Universal Robots PolyScope program: 1_dragon.urp

Program 1_dragon (installation=default directory=/programs/dragon_new createdIn=5.11.9.1010452 lastSavedIn=5.11.9.1010452 robotSerialNumber=20225200364)
Calibrated DH parameters: a=[0.00002, -0.569483, -0.54992, -0.00001, -0.000036, 0]; d=[0.180894, -146.691669, 192.918669, -46.053088, 0.119778, 0.115602]; alpha=[1.571425, -0.001534, 0.003359, 1.568739, -1.571477, 0]; deltaTheta=[0, 0.376258, -0.101074, -0.275185, -0.000002, 0]
Robot Program (runOnlyOnce=false)
  Script file /programs/usbdisk/1/dragon_rotate/john_midlower_rotate.script
    | def azat_dragon_rotate():
    |   # Global parameters:
    |   global speed_ms    = 0.3
    |   global speed_rads  = 0.750
    |   global accel_mss   = 1.000
    |   global accel_radss = 1.200
    |   global blend_radius_m = 0.001
    |   global ref_frame = p[0,0,0,0,0,0]
    | 
    |   #
    |   # TO REMOVE HEADER:
    |   # Go to "Program" -> "Post-Processor Editor"
    |   # Select "Universal Robots"
    |   # Set "INCLUDE_HEADER" to "False"
    |   #
    |   #--------------------------
    |   # Add any default subprograms here
    |   # For example, to drive a gripper as a program call:
    |   # def Gripper_Open():
    |   #   ...
    |   # end
    |   #
    |   # Example to drive a spray gun:
    |   def SprayOn(value):
    |     # use the value as an output:
    |     DO_SPRAY = 5
    |     if value == 0:
    |       set_standard_digital_out(DO_SPRAY, False)
    |     else:
    |       set_standard_digital_out(DO_SPRAY, True)
    |     end
    |   end
    | 
    |   # Example to drive an extruder:
    |   def Extruder(value):
    |     # use the value as an output:
    |     if value < 0:
    |       # stop extruder
    |     else:
    |       # start extruder
    |     end
    |   end
    | 
    |   # Example to move an external axis
    |   def MoveAxis(value):
    |     # use the value as an output:
    |     DO_AXIS_1 = 1
    |     DI_AXIS_1 = 1
    |     if value <= 0:
    |       set_standard_digital_out(DO_AXIS_1, False)
    | 
    |       # Wait for digital input to change state
    |       #while (get_standard_digital_in(DI_AXIS_1) != False):
    |       #  sync()
    |       #end
    |     else:
    |       set_standard_digital_out(DO_AXIS_1, True)
    | 
    |       # Wait for digital input to change state
    |       #while (get_standard_digital_in(DI_AXIS_1) != True):
    |       #  sync()
    |       #end
    |     end
    |   end
    |   #--------------------------
    | 
    | 
    |   # Main program:
    |   # Program generated by RoboDK v5.7.4 for UR10e on 14/08/2024 10:25:34
    |   # Using nominal kinematics.
    |   blend_radius_m = 0.001
    |   speed_ms    = 1.000
    |   ref_frame = p[0.339429, -0.052043, 0.008200, 0.000000, 0.000000, 0.000000]
    |   set_tcp(p[0.000000, 0.000000, 0.252000, 0.000000, 0.000000, 0.000000])
    |   # Show Tool
    |   movej([0.421631, -1.076921, -2.495001, -1.140464, 1.570796, 1.992433],accel_radss,speed_rads,0,0)
    |   movel(pose_trans(ref_frame,p[0.050000, 0.035848, 0.005000, -0.000000, 3.141593, -0.000000]),accel_mss,speed_ms,0,0) # end trace
    |   speed_ms    = 0.002
    |   movel(pose_trans(ref_frame,p[0.050000, 0.035848, -0.000125, -0.000000, 3.141593, -0.000000]),accel_mss,speed_ms,0,0) # end trace
    |   speed_ms    = 0.007
    |   movel(pose_trans(ref_frame,p[0.048115, 0.040844, -0.000125, 0.000000, 3.141593, 0.000000]),accel_mss,speed_ms,0,0.001)
    |   movel(pose_trans(ref_frame,p[0.048793, 0.046214, -0.000125, -0.000000, 3.141593, -0.000000]),accel_mss,speed_ms,0,0.001)
    |   movel(pose_trans(ref_frame,p[0.049357, 0.045822, -0.000125, -0.000000, 3.141593, -0.000000]),accel_mss,speed_ms,0,0.001)
    |   movel(pose_trans(ref_frame,p[0.050418, 0.046022, -0.000125, 0.000000, 3.141593, -0.000000]),accel_mss,speed_ms,0,0.001)
    |   movel(pose_trans(ref_frame,p[0.050476, 0.047250, -0.000125, 0.000000, 3.141593, -0.000000]),accel_mss,speed_ms,0,0.001)
    |   movel(pose_trans(ref_frame,p[0.050281, 0.048486, -0.000125, -0.000000, 3.141593, -0.000000]),accel_mss,speed_ms,0,0.001)
    |   movel(pose_trans(ref_frame,p[0.050801, 0.052016, -0.000125, -0.000000, 3.141593, -0.000000]),accel_mss,speed_ms,0,0.001)
    |   movel(pose_trans(ref_frame,p[0.052856, 0.054981, -0.000125, 0.000000, 3.141593, -0.000000]),accel_mss,speed_ms,0,0.001)
    |   movel(pose_trans(ref_frame,p[0.052477, 0.053383, -0.000125, 0.000000, 3.141593, -0.000000]),accel_mss,speed_ms,0,0.001)
    |   movel(pose_trans(ref_frame,p[0.053030, 0.051842, -0.000125, 0.000000, 3.141593, 0.000000]),accel_mss,speed_ms,0,0.001)
    |   movel(pose_trans(ref_frame,p[0.053222, 0.051718, -0.000125, 0.000000, 3.141593, -0.000000]),accel_mss,speed_ms,0,0.001)
    |   movel(pose_trans(ref_frame,p[0.053441, 0.051660, -0.000125, 0.000000, 3.141593, -0.000000]),accel_mss,speed_ms,0,0.001)
    |   movel(pose_trans(ref_frame,p[0.053830, 0.051770, -0.000125, -0.000000, 3.141593, -0.000000]),accel_mss,speed_ms,0,0.001)
    |   movel(pose_trans(ref_frame,p[0.054167, 0.052030, -0.000125, 0.000000, 3.141593, 0.000000]),accel_mss,speed_ms,0,0.001)
    |   movel(pose_trans(ref_frame,p[0.057601, 0.053765, -0.000125, 0.000000, 3.141593, -0.000000]),accel_mss,speed_ms,0,0.001)
    |   movel(pose_trans(ref_frame,p[0.061373, 0.053375, -0.000125, 0.000000, 3.141593, -0.000000]),accel_mss,speed_ms,0,0.001)
    |   movel(pose_trans(ref_frame,p[0.059629, 0.053360, -0.000125, -0.000000, 3.141593, -0.000000]),accel_mss,speed_ms,0,0.001)
    |   movel(pose_trans(ref_frame,p[0.058435, 0.051934, -0.000125, -0.000000, 3.141593, -0.000000]),accel_mss,speed_ms,0,0.001)
    |   movel(pose_trans(ref_frame,p[0.058753, 0.051481, -0.000125, -0.000000, 3.141593, -0.000000]),accel_mss,speed_ms,0,0.001)
    |   movel(pose_trans(ref_frame,p[0.059332, 0.051255, -0.000125, 0.000000, 3.141593, -0.000000]),accel_mss,speed_ms,0,0.001)
    |   movel(pose_trans(ref_frame,p[0.063602, 0.049837, -0.000125, -0.000000, 3.141593, -0.000000]),accel_mss,speed_ms,0,0.001)
    |   movel(pose_trans(ref_frame,p[0.067592, 0.047737, -0.000125, -0.000000, 3.141593, 0.000000]),accel_mss,speed_ms,0,0.001)
    |   movel(pose_trans(ref_frame,p[0.066591, 0.047674, -0.000125, -0.000000, 3.141593, 0.000000]),accel_mss,speed_ms,0,0.001)
    |   movel(pose_trans(ref_frame,p[0.065618, 0.047434, -0.000125, 0.000000, 3.141593, -0.000000]),accel_mss,speed_ms,0,0.001)
    |   movel(pose_trans(ref_frame,p[0.065188, 0.047247, -0.000125, -0.000000, 3.141593, 0.000000]),accel_mss,speed_ms,0,0.001)
    |   movel(pose_trans(ref_frame,p[0.064838, 0.046949, -0.000125, 0.000000, 3.141593, -0.000000]),accel_mss,speed_ms,0,0.001)
    |   movel(pose_trans(ref_frame,p[0.065795, 0.044806, -0.000125, -0.000000, 3.141593, 0.000000]),accel_mss,speed_ms,0,0.001)
    |   movel(pose_trans(ref_frame,p[0.068800, 0.043786, -0.000125, -0.000000, 3.141593, 0.000000]),accel_mss,speed_ms,0,0.001)
    |   movel(pose_trans(ref_frame,p[0.071196, 0.042031, -0.000125, -0.000000, 3.141593, -0.000000]),accel_mss,speed_ms,0,0.001)
    |   movel(pose_trans(ref_frame,p[0.073265, 0.039897, -0.000125, 0.000000, 3.141593, -0.000000]),accel_mss,speed_ms,0,0.001)
    |   movel(pose_trans(ref_frame,p[0.072103, 0.040443, -0.000125, 0.000000, 3.141593, 0.000000]),accel_mss,speed_ms,0,0.001)
    |   movel(pose_trans(ref_frame,p[0.070839, 0.040620, -0.000125, -0.000000, 3.141593, 0.000000]),accel_mss,speed_ms,0,0.001)
    |   movel(pose_trans(ref_frame,p[0.070205, 0.040771, -0.000125, 0.000000, 3.141593, -0.000000]),accel_mss,speed_ms,0,0.001)
    |   movel(pose_trans(ref_frame,p[0.069592, 0.040656, -0.000125, -0.000000, 3.141593, -0.000000]),accel_mss,speed_ms,0,0.001)
    |   movel(pose_trans(ref_frame,p[0.069908, 0.038813, -0.000125, -0.000000, 3.141593, 0.000000]),accel_mss,speed_ms,0,0.001)
    |   movel(pose_trans(ref_frame,p[0.071559, 0.038089, -0.000125, -0.000000, 3.141593, -0.000000]),accel_mss,speed_ms,0,0.001)
    |   movel(pose_trans(ref_frame,p[0.074165, 0.036670, -0.000125, -0.000000, 3.141593, 0.000000]),accel_mss,speed_ms,0,0.001)
    |   movel(pose_trans(ref_frame,p[0.076688, 0.035073, -0.000125, -0.000000, 3.141593, -0.000000]),accel_mss,speed_ms,0,0.001)
    |   movel(pose_trans(ref_frame,p[0.077386, 0.034559, -0.000125, -0.000000, 3.141593, -0.000000]),accel_mss,speed_ms,0,0.001)
    |   movel(pose_trans(ref_frame,p[0.077983, 0.033940, -0.000125, -0.000000, 3.141593, -0.000000]),accel_mss,speed_ms,0,0.001)
    |   movel(pose_trans(ref_frame,p[0.078075, 0.033778, -0.000125, 0.000000, 3.141593, -0.000000]),accel_mss,speed_ms,0,0.001)
    |   movel(pose_trans(ref_frame,p[0.078069, 0.033607, -0.000125, -0.000000, 3.141593, -0.000000]),accel_mss,speed_ms,0,0.001)
    |   movel(pose_trans(ref_frame,p[0.075726, 0.034474, -0.000125, -0.000000, 3.141593, -0.000000]),accel_mss,speed_ms,0,0.001)
    |   movel(pose_trans(ref_frame,p[0.073247, 0.033725, -0.000125, 0.000000, 3.141593, 0.000000]),accel_mss,speed_ms,0,0.001)
    |   movel(pose_trans(ref_frame,p[0.073124, 0.033569, -0.000125, -0.000000, 3.141593, -0.000000]),accel_mss,speed_ms,0,0.001)
    |   movel(pose_trans(ref_frame,p[0.073061, 0.033386, -0.000125, -0.000000, 3.141593, -0.000000]),accel_mss,speed_ms,0,0.001)
    |   movel(pose_trans(ref_frame,p[0.073215, 0.033032, -0.000125, -0.000000, 3.141593, -0.000000]),accel_mss,speed_ms,0,0.001)
    |   movel(pose_trans(ref_frame,p[0.073585, 0.032804, -0.000125, -0.000000, 3.141593, -0.000000]),accel_mss,speed_ms,0,0.001)
    |   movel(pose_trans(ref_frame,p[0.077970, 0.030799, -0.000125, 0.000000, 3.141593, -0.000000]),accel_mss,speed_ms,0,0.001)
    |   movel(pose_trans(ref_frame,p[0.081965, 0.028072, -0.000125, -0.000000, 3.141593, 0.000000]),accel_mss,speed_ms,0,0.001)
    |   movel(pose_trans(ref_frame,p[0.080851, 0.028334, -0.000125, -0.000000, 3.141593, -0.000000]),accel_mss,speed_ms,0,0.001)
    |   movel(pose_trans(ref_frame,p[0.079709, 0.028175, -0.000125, -0.000000, 3.141593, 0.000000]),accel_mss,speed_ms,0,0.001)
    |   movel(pose_trans(ref_frame,p[0.079538, 0.027599, -0.000125, 0.000000, 3.141593, -0.000000]),accel_mss,speed_ms,0,0.001)
    |   movel(pose_trans(ref_frame,p[0.080054, 0.027314, -0.000125, -0.000000, 3.141593, 0.000000]),accel_mss,speed_ms,0,0.001)
    |   movel(pose_trans(ref_frame,p[0.081649, 0.027083, -0.000125, 0.000000, 3.141593, -0.000000]),accel_mss,speed_ms,0,0.001)
    |   movel(pose_trans(ref_frame,p[0.083244, 0.026828, -0.000125, 0.000000, 3.141593, 0.000000]),accel_mss,speed_ms,0,0.001)
    |   movel(pose_trans(ref_frame,p[0.085130, 0.026266, -0.000125, -0.000000, 3.141593, -0.000000]),accel_mss,speed_ms,0,0.001)
    |   movel(pose_trans(ref_frame,p[0.086815, 0.025298, -0.000125, -0.000000, 3.141593, -0.000000]),accel_mss,speed_ms,0,0.001)
    |   movel(pose_trans(ref_frame,p[0.085082, 0.025169, -0.000125, -0.000000, 3.141593, -0.000000]),accel_mss,speed_ms,0,0.001)
    |   movel(pose_trans(ref_frame,p[0.083511, 0.024408, -0.000125, -0.000000, 3.141593, -0.000000]),accel_mss,speed_ms,0,0.001)
    |   movel(pose_trans(ref_frame,p[0.084423, 0.023039, -0.000125, -0.000000, 3.141593, -0.000000]),accel_mss,speed_ms,0,0.001)
    |   movel(pose_trans(ref_frame,p[0.086438, 0.023247, -0.000125, -0.000000, 3.141593, -0.000000]),accel_mss,speed_ms,0,0.001)
    |   movel(pose_trans(ref_frame,p[0.087631, 0.023229, -0.000125, -0.000000, 3.141593, -0.000000]),accel_mss,speed_ms,0,0.001)
    |   movel(pose_trans(ref_frame,p[0.088824, 0.023201, -0.000125, 0.000000, 3.141593, 0.000000]),accel_mss,speed_ms,0,0.001)
    |   movel(pose_trans(ref_frame,p[0.090324, 0.022840, -0.000125, 0.000000, 3.141593, -0.000000]),accel_mss,speed_ms,0,0.001)
    |   movel(pose_trans(ref_frame,p[0.091725, 0.022190, -0.000125, -0.000000, 3.141593, -0.000000]),accel_mss,speed_ms,0,0.001)
    |   movel(pose_trans(ref_frame,p[0.090634, 0.022048, -0.000125, -0.000000, 3.141593, -0.000000]),accel_mss,speed_ms,0,0.001)
    |   movel(pose_trans(ref_frame,p[0.089714, 0.021514, -0.000125, -0.000000, 3.141593, -0.000000]),accel_mss,speed_ms,0,0.001)
    |   movel(pose_trans(ref_frame,p[0.089568, 0.021326, -0.000125, -0.000000, 3.141593, -0.000000]),accel_mss,speed_ms,0,0.001)
    |   movel(pose_trans(ref_frame,p[0.089490, 0.021107, -0.000125, 0.000000, 3.141593, -0.000000]),accel_mss,speed_ms,0,0.001)
    |   movel(pose_trans(ref_frame,p[0.089956, 0.020148, -0.000125, -0.000000, 3.141593, 0.000000]),accel_mss,speed_ms,0,0.001)
    |   movel(pose_trans(ref_frame,p[0.090905, 0.019837, -0.000125, -0.000000, 3.141593, -0.000000]),accel_mss,speed_ms,0,0.001)
    |   movel(pose_trans(ref_frame,p[0.093609, 0.020103, -0.000125, -0.000000, 3.141593, -0.000000]),accel_mss,speed_ms,0,0.001)
    |   movel(pose_trans(ref_frame,p[0.096074, 0.021219, -0.000125, -0.000000, 3.141593, -0.000000]),accel_mss,speed_ms,0,0.001)
    |   movel(pose_trans(ref_frame,p[0.095278, 0.019985, -0.000125, -0.000000, 3.141593, -0.000000]),accel_mss,speed_ms,0,0.001)
    |   movel(pose_trans(ref_frame,p[0.096057, 0.018680, -0.000125, 0.000000, 3.141593, 0.000000]),accel_mss,speed_ms,0,0.001)
    |   movel(pose_trans(ref_frame,p[0.097535, 0.018934, -0.000125, -0.000000, 3.141593, 0.000000]),accel_mss,speed_ms,0,0.001)
    |   movel(pose_trans(ref_frame,p[0.098790, 0.019781, -0.000125, 0.000000, 3.141593, -0.000000]),accel_mss,speed_ms,0,0.001)
    |   movel(pose_trans(ref_frame,p[0.100083, 0.020616, -0.000125, 0.000000, 3.141593, -0.000000]),accel_mss,speed_ms,0,0.001)
    |   movel(pose_trans(ref_frame,p[0.101189, 0.021687, -0.000125, -0.000000, 3.141593, -0.000000]),accel_mss,speed_ms,0,0.001)
    |   movel(pose_trans(ref_frame,p[0.101202, 0.020923, -0.000125, -0.000000, 3.141593, -0.000000]),accel_mss,speed_ms,0,0.001)
    |   movel(pose_trans(ref_frame,p[0.101280, 0.020162, -0.000125, -0.000000, 3.141593, -0.000000]),accel_mss,speed_ms,0,0.001)
    |   movel(pose_trans(ref_frame,p[0.101434, 0.019617, -0.000125, -0.000000, 3.141593, 0.000000]),accel_mss,speed_ms,0,0.001)
    |   movel(pose_trans(ref_frame,p[0.101820, 0.019279, -0.000125, -0.000000, 3.141593, 0.000000]),accel_mss,speed_ms,0,0.001)
    |   movel(pose_trans(ref_frame,p[0.103405, 0.020161, -0.000125, -0.000000, 3.141593, -0.000000]),accel_mss,speed_ms,0,0.001)
    |   movel(pose_trans(ref_frame,p[0.103922, 0.021711, -0.000125, -0.000000, 3.141593, 0.000000]),accel_mss,speed_ms,0,0.001)
    |   movel(pose_trans(ref_frame,p[0.104603, 0.023835, -0.000125, -0.000000, 3.141593, 0.000000]),accel_mss,speed_ms,0,0.001)
    |   movel(pose_trans(ref_frame,p[0.105672, 0.025813, -0.000125, 0.000000, 3.141593, -0.000000]),accel_mss,speed_ms,0,0.001)
    |   movel(pose_trans(ref_frame,p[0.106210, 0.023998, -0.000125, 0.000000, 3.141593, -0.000000]),accel_mss,speed_ms,0,0.001)
    |   movel(pose_trans(ref_frame,p[0.106813, 0.023627, -0.000125, -0.000000, 3.141593, 0.000000]),accel_mss,speed_ms,0,0.001)
    |   movel(pose_trans(ref_frame,p[0.107376, 0.023906, -0.000125, 0.000000, 3.141593, 0.000000]),accel_mss,speed_ms,0,0.001)
    |   movel(pose_trans(ref_frame,p[0.107881, 0.025705, -0.000125, -0.000000, 3.141593, -0.000000]),accel_mss,speed_ms,0,0.001)
    |   movel(pose_trans(ref_frame,p[0.107658, 0.028092, -0.000125, -0.000000, 3.141593, -0.000000]),accel_mss,speed_ms,0,0.001)
    |   movel(pose_trans(ref_frame,p[0.107800, 0.030579, -0.000125, -0.000000, 3.141593, -0.000000]),accel_mss,speed_ms,0,0.001)
    |   movel(pose_trans(ref_frame,p[0.109047, 0.029228, -0.000125, -0.000000, 3.141593, -0.000000]),accel_mss,speed_ms,0,0.001)
    |   movel(pose_trans(ref_frame,p[0.110204, 0.030182, -0.000125, -0.000000, 3.141593, -0.000000]),accel_mss,speed_ms,0,0.001)
    |   movel(pose_trans(ref_frame,p[0.109002, 0.033200, -0.000125, -0.000000, 3.141593, -0.000000]),accel_mss,speed_ms,0,0.001)
    |   movel(pose_trans(ref_frame,p[0.107979, 0.036132, -0.000125, -0.000000, 3.141593, 0.000000]),accel_mss,speed_ms,0,0.001)
    |   movel(pose_trans(ref_frame,p[0.108895, 0.035281, -0.000125, -0.000000, 3.141593, -0.000000]),accel_mss,speed_ms,0,0.001)
    |   movel(pose_trans(ref_frame,p[0.110237, 0.035493, -0.000125, -0.000000, 3.141593, -0.000000]),accel_mss,speed_ms,0,0.001)
    |   movel(pose_trans(ref_frame,p[0.110068, 0.037051, -0.000125, 0.000000, 3.141593, 0.000000]),accel_mss,speed_ms,0,0.001)
    |   movel(pose_trans(ref_frame,p[0.109162, 0.038243, -0.000125, -0.000000, 3.141593, -0.000000]),accel_mss,speed_ms,0,0.001)
    |   movel(pose_trans(ref_frame,p[0.108731, 0.039432, -0.000125, 0.000000, 3.141593, -0.000000]),accel_mss,speed_ms,0,0.001)
    |   movel(pose_trans(ref_frame,p[0.108673, 0.040695, -0.000125, 0.000000, 3.141593, -0.000000]),accel_mss,speed_ms,0,0) # end trace
    |   speed_ms    = 1.000
    |   movel(pose_trans(ref_frame,p[0.108673, 0.040695, 0.005000, 0.000000, 3.141593, -0.000000]),accel_mss,speed_ms,0,0.001)
    |   movel(pose_trans(ref_frame,p[0.105336, 0.049069, 0.005000, 0.000000, 3.141593, -0.000000]),accel_mss,speed_ms,0,0) # end trace
    |   speed_ms    = 0.002
    |   movel(pose_trans(ref_frame,p[0.105336, 0.049069, -0.000125, 0.000000, 3.141593, 0.000000]),accel_mss,speed_ms,0,0) # end trace
    |   speed_ms    = 0.007
    |   movel(pose_trans(ref_frame,p[0.100848, 0.047278, -0.000125, 0.000000, 3.141593, -0.000000]),accel_mss,speed_ms,0,0.001)
    |   movel(pose_trans(ref_frame,p[0.096181, 0.046825, -0.000125, -0.000000, 3.141593, -0.000000]),accel_mss,speed_ms,0,0.001)
    |   movel(pose_trans(ref_frame,p[0.092012, 0.048769, -0.000125, -0.000000, 3.141593, 0.000000]),accel_mss,speed_ms,0,0.001)
    |   movel(pose_trans(ref_frame,p[0.090230, 0.052991, -0.000125, -0.000000, 3.141593, 0.000000]),accel_mss,speed_ms,0,0.001)
    |   movel(pose_trans(ref_frame,p[0.090956, 0.059068, -0.000125, -0.000000, 3.141593, -0.000000]),accel_mss,speed_ms,0,0.001)
    |   movel(pose_trans(ref_frame,p[0.093240, 0.064896, -0.000125, -0.000000, 3.141593, -0.000000]),accel_mss,speed_ms,0,0.001)
    |   movel(pose_trans(ref_frame,p[0.093396, 0.065125, -0.000125, -0.000000, 3.141593, -0.000000]),accel_mss,speed_ms,0,0.001)
    |   movel(pose_trans(ref_frame,p[0.093608, 0.065293, -0.000125, -0.000000, 3.141593, -0.000000]),accel_mss,speed_ms,0,0.001)
    |   movel(pose_trans(ref_frame,p[0.094176, 0.065243, -0.000125, -0.000000, 3.141593, -0.000000]),accel_mss,speed_ms,0,0.001)
    |   movel(pose_trans(ref_frame,p[0.094662, 0.064808, -0.000125, 0.000000, 3.141593, 0.000000]),accel_mss,speed_ms,0,0.001)
    |   movel(pose_trans(ref_frame,p[0.095614, 0.063660, -0.000125, 0.000000, 3.141593, 0.000000]),accel_mss,speed_ms,0,0.001)
    |   movel(pose_trans(ref_frame,p[0.100924, 0.056746, -0.000125, 0.000000, 3.141593, -0.000000]),accel_mss,speed_ms,0,0.001)
    |   movel(pose_trans(ref_frame,p[0.105953, 0.049801, -0.000125, -0.000000, 3.141593, -0.000000]),accel_mss,speed_ms,0,0.001)
    |   movel(pose_trans(ref_frame,p[0.105818, 0.049295, -0.000125, 0.000000, 3.141593, 0.000000]),accel_mss,speed_ms,0,0.001)
    |   movel(pose_trans(ref_frame,p[0.105578, 0.049182, -0.000125, -0.000000, 3.141593, -0.000000]),accel_mss,speed_ms,0,0.001)
    |   movel(pose_trans(ref_frame,p[0.105336, 0.049069, -0.000125, 0.000000, 3.141593, 0.000000]),accel_mss,speed_ms,0,0) # end trace
    |   speed_ms    = 1.000
    |   movel(pose_trans(ref_frame,p[0.105336, 0.049069, 0.005000, 0.000000, 3.141593, -0.000000]),accel_mss,speed_ms,0,0.001)
    |   movel(pose_trans(ref_frame,p[0.089633, 0.087186, 0.005000, -0.000000, 3.141593, 0.000000]),accel_mss,speed_ms,0,0) # end trace
    |   speed_ms    = 0.002
    |   movel(pose_trans(ref_frame,p[0.089633, 0.087186, -0.000125, -0.000000, 3.141593, -0.000000]),accel_mss,speed_ms,0,0) # end trace
    |   speed_ms    = 0.007
    |   movel(pose_trans(ref_frame,p[0.091088, 0.088696, -0.000125, -0.000000, 3.141593, 0.000000]),accel_mss,speed_ms,0,0.001)
    |   movel(pose_trans(ref_frame,p[0.092593, 0.090142, -0.000125, 0.000000, 3.141593, 0.000000]),accel_mss,speed_ms,0,0.001)
    |   movel(pose_trans(ref_frame,p[0.093893, 0.091163, -0.000125, 0.000000, 3.141593, 0.000000]),accel_mss,speed_ms,0,0.001)
    |   movel(pose_trans(ref_frame,p[0.095145, 0.092291, -0.000125, -0.000000, 3.141593, 0.000000]),accel_mss,speed_ms,0,0.001)
    |   movel(pose_trans(ref_frame,p[0.096993, 0.095273, -0.000125, -0.000000, 3.141593, 0.000000]),accel_mss,speed_ms,0,0.001)
    |   movel(pose_trans(ref_frame,p[0.098237, 0.098544, -0.000125, -0.000000, 3.141593, 0.000000]),accel_mss,speed_ms,0,0.001)
    |   movel(pose_trans(ref_frame,p[0.098481, 0.099687, -0.000125, 0.000000, 3.141593, -0.000000]),accel_mss,speed_ms,0,0.001)
    |   movel(pose_trans(ref_frame,p[0.098141, 0.100704, -0.000125, -0.000000, 3.141593, -0.000000]),accel_mss,speed_ms,0,0.001)
    |   movel(pose_trans(ref_frame,p[0.097842, 0.100958, -0.000125, -0.000000, 3.141593, -0.000000]),accel_mss,speed_ms,0,0.001)
    |   movel(pose_trans(ref_frame,p[0.097539, 0.101210, -0.000125, 0.000000, 3.141593, 0.000000]),accel_mss,speed_ms,0,0.001)
    |   movel(pose_trans(ref_frame,p[0.097169, 0.102392, -0.000125, 0.000000, 3.141593, -0.000000]),accel_mss,speed_ms,0,0.001)
    |   movel(pose_trans(ref_frame,p[0.097527, 0.103718, -0.000125, -0.000000, 3.141593, 0.000000]),accel_mss,speed_ms,0,0.001)
    |   movel(pose_trans(ref_frame,p[0.096297, 0.103890, -0.000125, -0.000000, 3.141593, 0.000000]),accel_mss,speed_ms,0,0.001)
    |   movel(pose_trans(ref_frame,p[0.095148, 0.103405, -0.000125, -0.000000, 3.141593, -0.000000]),accel_mss,speed_ms,0,0.001)
    |   movel(pose_trans(ref_frame,p[0.093699, 0.102652, -0.000125, 0.000000, 3.141593, 0.000000]),accel_mss,speed_ms,0,0.001)
    |   movel(pose_trans(ref_frame,p[0.092339, 0.101738, -0.000125, -0.000000, 3.141593, 0.000000]),accel_mss,speed_ms,0,0.001)
    |   movel(pose_trans(ref_frame,p[0.084495, 0.094077, -0.000125, 0.000000, 3.141593, -0.000000]),accel_mss,speed_ms,0,0.001)
    |   movel(pose_trans(ref_frame,p[0.078491, 0.084897, -0.000125, -0.000000, 3.141593, 0.000000]),accel_mss,speed_ms,0,0.001)
    |   movel(pose_trans(ref_frame,p[0.076525, 0.081104, -0.000125, 0.000000, 3.141593, 0.000000]),accel_mss,speed_ms,0,0.001)
    |   movel(pose_trans(ref_frame,p[0.074922, 0.077142, -0.000125, -0.000000, 3.141593, -0.000000]),accel_mss,speed_ms,0,0.001)
    |   movel(pose_trans(ref_frame,p[0.074131, 0.071003, -0.000125, -0.000000, 3.141593, -0.000000]),accel_mss,speed_ms,0,0.001)
    |   movel(pose_trans(ref_frame,p[0.072889, 0.069893, -0.000125, -0.000000, 3.141593, -0.000000]),accel_mss,speed_ms,0,0.001)
    |   movel(pose_trans(ref_frame,p[0.072797, 0.069931, -0.000125, 0.000000, 3.141593, -0.000000]),accel_mss,speed_ms,0,0.001)
    |   movel(pose_trans(ref_frame,p[0.072716, 0.069992, -0.000125, 0.000000, 3.141593, -0.000000]),accel_mss,speed_ms,0,0.001)
    |   movel(pose_trans(ref_frame,p[0.071475, 0.071671, -0.000125, -0.000000, 3.141593, -0.000000]),accel_mss,speed_ms,0,0.001)
    |   movel(pose_trans(ref_frame,p[0.070262, 0.073293, -0.000125, 0.000000, 3.141593, 0.000000]),accel_mss,speed_ms,0,0.001)
    |   movel(pose_trans(ref_frame,p[0.068510, 0.073911, -0.000125, 0.000000, 3.141593, 0.000000]),accel_mss,speed_ms,0,0.001)
    |   movel(pose_trans(ref_frame,p[0.066701, 0.073510, -0.000125, 0.000000, 3.141593, 0.000000]),accel_mss,speed_ms,0,0.001)
    |   movel(pose_trans(ref_frame,p[0.064031, 0.071756, -0.000125, 0.000000, 3.141593, 0.000000]),accel_mss,speed_ms,0,0.001)
    |   movel(pose_trans(ref_frame,p[0.061632, 0.069604, -0.000125, 0.000000, 3.141593, -0.000000]),accel_mss,speed_ms,0,0.001)
    |   movel(pose_trans(ref_frame,p[0.058330, 0.065115, -0.000125, -0.000000, 3.141593, -0.000000]),accel_mss,speed_ms,0,0.001)
    |   movel(pose_trans(ref_frame,p[0.057824, 0.059503, -0.000125, 0.000000, 3.141593, 0.000000]),accel_mss,speed_ms,0,0.001)
    |   movel(pose_trans(ref_frame,p[0.060086, 0.058641, -0.000125, 0.000000, 3.141593, 0.000000]),accel_mss,speed_ms,0,0.001)
    |   movel(pose_trans(ref_frame,p[0.062094, 0.060133, -0.000125, 0.000000, 3.141593, 0.000000]),accel_mss,speed_ms,0,0.001)
    |   movel(pose_trans(ref_frame,p[0.064267, 0.062034, -0.000125, 0.000000, 3.141593, -0.000000]),accel_mss,speed_ms,0,0.001)
    |   movel(pose_trans(ref_frame,p[0.066707, 0.063601, -0.000125, 0.000000, 3.141593, -0.000000]),accel_mss,speed_ms,0,0.001)
    |   movel(pose_trans(ref_frame,p[0.067317, 0.063786, -0.000125, -0.000000, 3.141593, -0.000000]),accel_mss,speed_ms,0,0.001)
    |   movel(pose_trans(ref_frame,p[0.067927, 0.063723, -0.000125, 0.000000, 3.141593, -0.000000]),accel_mss,speed_ms,0,0.001)
    |   movel(pose_trans(ref_frame,p[0.068318, 0.063438, -0.000125, -0.000000, 3.141593, -0.000000]),accel_mss,speed_ms,0,0.001)
    |   movel(pose_trans(ref_frame,p[0.068611, 0.063039, -0.000125, -0.000000, 3.141593, -0.000000]),accel_mss,speed_ms,0,0.001)
    |   movel(pose_trans(ref_frame,p[0.069511, 0.061129, -0.000125, 0.000000, 3.141593, -0.000000]),accel_mss,speed_ms,0,0.001)
    |   movel(pose_trans(ref_frame,p[0.070136, 0.059096, -0.000125, -0.000000, 3.141593, -0.000000]),accel_mss,speed_ms,0,0.001)
    |   movel(pose_trans(ref_frame,p[0.071200, 0.054465, -0.000125, -0.000000, 3.141593, 0.000000]),accel_mss,speed_ms,0,0.001)
    |   movel(pose_trans(ref_frame,p[0.072592, 0.049848, -0.000125, 0.000000, 3.141593, -0.000000]),accel_mss,speed_ms,0,0.001)
    |   movel(pose_trans(ref_frame,p[0.074780, 0.046144, -0.000125, -0.000000, 3.141593, -0.000000]),accel_mss,speed_ms,0,0.001)
    |   movel(pose_trans(ref_frame,p[0.078924, 0.047029, -0.000125, -0.000000, 3.141593, -0.000000]),accel_mss,speed_ms,0,0.001)
    |   movel(pose_trans(ref_frame,p[0.078996, 0.048255, -0.000125, 0.000000, 3.141593, 0.000000]),accel_mss,speed_ms,0,0.001)
    |   movel(pose_trans(ref_frame,p[0.078814, 0.049489, -0.000125, -0.000000, 3.141593, -0.000000]),accel_mss,speed_ms,0,0.001)
    |   movel(pose_trans(ref_frame,p[0.079748, 0.069610, -0.000125, -0.000000, 3.141593, -0.000000]),accel_mss,speed_ms,0,0.001)
    |   movel(pose_trans(ref_frame,p[0.089629, 0.087186, -0.000125, 0.000000, 3.141593, 0.000000]),accel_mss,speed_ms,0,0) # end trace
    |   speed_ms    = 1.000
    |   movel(pose_trans(ref_frame,p[0.089633, 0.087186, 0.005000, -0.000000, 3.141593, 0.000000]),accel_mss,speed_ms,0,0.001)
    |   movel(pose_trans(ref_frame,p[0.102749, 0.098109, 0.005000, 0.000000, 3.141593, -0.000000]),accel_mss,speed_ms,0,0) # end trace
    |   speed_ms    = 0.002
    |   movel(pose_trans(ref_frame,p[0.102749, 0.098109, -0.000125, 0.000000, 3.141593, -0.000000]),accel_mss,speed_ms,0,0) # end trace
    |   speed_ms    = 0.007
    |   movel(pose_trans(ref_frame,p[0.100717, 0.101702, -0.000125, 0.000000, 3.141593, 0.000000]),accel_mss,speed_ms,0,0.001)
    |   movel(pose_trans(ref_frame,p[0.100054, 0.105778, -0.000125, 0.000000, 3.141593, -0.000000]),accel_mss,speed_ms,0,0.001)
    |   movel(pose_trans(ref_frame,p[0.100478, 0.105179, -0.000125, -0.000000, 3.141593, 0.000000]),accel_mss,speed_ms,0,0.001)
    |   movel(pose_trans(ref_frame,p[0.100830, 0.104483, -0.000125, 0.000000, 3.141593, -0.000000]),accel_mss,speed_ms,0,0.001)
    |   movel(pose_trans(ref_frame,p[0.103117, 0.102032, -0.000125, -0.000000, 3.141593, 0.000000]),accel_mss,speed_ms,0,0.001)
    |   movel(pose_trans(ref_frame,p[0.106032, 0.100361, -0.000125, -0.000000, 3.141593, 0.000000]),accel_mss,speed_ms,0,0.001)
    |   movel(pose_trans(ref_frame,p[0.107531, 0.101698, -0.000125, -0.000000, 3.141593, -0.000000]),accel_mss,speed_ms,0,0.001)
    |   movel(pose_trans(ref_frame,p[0.106753, 0.104177, -0.000125, -0.000000, 3.141593, 0.000000]),accel_mss,speed_ms,0,0.001)
    |   movel(pose_trans(ref_frame,p[0.107988, 0.102605, -0.000125, 0.000000, 3.141593, 0.000000]),accel_mss,speed_ms,0,0.001)
    |   movel(pose_trans(ref_frame,p[0.109319, 0.101130, -0.000125, -0.000000, 3.141593, 0.000000]),accel_mss,speed_ms,0,0.001)
    |   movel(pose_trans(ref_frame,p[0.112898, 0.098528, -0.000125, -0.000000, 3.141593, 0.000000]),accel_mss,speed_ms,0,0.001)
    |   movel(pose_trans(ref_frame,p[0.116000, 0.095504, -0.000125, -0.000000, 3.141593, 0.000000]),accel_mss,speed_ms,0,0.001)
    |   movel(pose_trans(ref_frame,p[0.115507, 0.097438, -0.000125, -0.000000, 3.141593, 0.000000]),accel_mss,speed_ms,0,0.001)
    |   movel(pose_trans(ref_frame,p[0.114821, 0.099297, -0.000125, 0.000000, 3.141593, -0.000000]),accel_mss,speed_ms,0,0.001)
    |   movel(pose_trans(ref_frame,p[0.116243, 0.097691, -0.000125, 0.000000, 3.141593, -0.000000]),accel_mss,speed_ms,0,0.001)
    |   movel(pose_trans(ref_frame,p[0.117809, 0.096208, -0.000125, 0.000000, 3.141593, -0.000000]),accel_mss,speed_ms,0,0.001)
    |   movel(pose_trans(ref_frame,p[0.119446, 0.093932, -0.000125, 0.000000, 3.141593, -0.000000]),accel_mss,speed_ms,0,0.001)
    |   movel(pose_trans(ref_frame,p[0.120874, 0.091548, -0.000125, 0.000000, 3.141593, 0.000000]),accel_mss,speed_ms,0,0.001)
    |   movel(pose_trans(ref_frame,p[0.121474, 0.090885, -0.000125, 0.000000, 3.141593, -0.000000]),accel_mss,speed_ms,0,0.001)
    |   movel(pose_trans(ref_frame,p[0.122260, 0.090597, -0.000125, -0.000000, 3.141593, 0.000000]),accel_mss,speed_ms,0,0.001)
    |   movel(pose_trans(ref_frame,p[0.123089, 0.090981, -0.000125, 0.000000, 3.141593, -0.000000]),accel_mss,speed_ms,0,0.001)
    |   movel(pose_trans(ref_frame,p[0.123661, 0.091788, -0.000125, 0.000000, 3.141593, -0.000000]),accel_mss,speed_ms,0,0.001)
    |   movel(pose_trans(ref_frame,p[0.124539, 0.088269, -0.000125, -0.000000, 3.141593, 0.000000]),accel_mss,speed_ms,0,0.001)
    |   movel(pose_trans(ref_frame,p[0.125564, 0.084887, -0.000125, -0.000000, 3.141593, -0.000000]),accel_mss,speed_ms,0,0.001)
    |   movel(pose_trans(ref_frame,p[0.125556, 0.082021, -0.000125, -0.000000, 3.141593, 0.000000]),accel_mss,speed_ms,0,0.001)
    |   movel(pose_trans(ref_frame,p[0.124836, 0.079246, -0.000125, -0.000000, 3.141593, -0.000000]),accel_mss,speed_ms,0,0) # end trace
    |   speed_ms    = 1.000
    |   movel(pose_trans(ref_frame,p[0.124836, 0.079246, 0.005000, -0.000000, 3.141593, 0.000000]),accel_mss,speed_ms,0,0.001)
    |   movel(pose_trans(ref_frame,p[0.070961, 0.083800, 0.005000, -0.000000, 3.141593, -0.000000]),accel_mss,speed_ms,0,0) # end trace
    |   speed_ms    = 0.002
    |   movel(pose_trans(ref_frame,p[0.070961, 0.083800, -0.000125, -0.000000, 3.141593, -0.000000]),accel_mss,speed_ms,0,0) # end trace
    |   speed_ms    = 0.007
    |   movel(pose_trans(ref_frame,p[0.069945, 0.082016, -0.000125, -0.000000, 3.141593, -0.000000]),accel_mss,speed_ms,0,0.001)
    |   movel(pose_trans(ref_frame,p[0.068221, 0.080903, -0.000125, -0.000000, 3.141593, -0.000000]),accel_mss,speed_ms,0,0.001)
    |   movel(pose_trans(ref_frame,p[0.062416, 0.082363, -0.000125, 0.000000, 3.141593, -0.000000]),accel_mss,speed_ms,0,0.001)
    |   movel(pose_trans(ref_frame,p[0.059213, 0.087150, -0.000125, 0.000000, 3.141593, 0.000000]),accel_mss,speed_ms,0,0.001)
    |   movel(pose_trans(ref_frame,p[0.057492, 0.092576, -0.000125, 0.000000, 3.141593, 0.000000]),accel_mss,speed_ms,0,0.001)
    |   movel(pose_trans(ref_frame,p[0.056740, 0.098209, -0.000125, -0.000000, 3.141593, 0.000000]),accel_mss,speed_ms,0,0.001)
    |   movel(pose_trans(ref_frame,p[0.056549, 0.100188, -0.000125, -0.000000, 3.141593, -0.000000]),accel_mss,speed_ms,0,0.001)
    |   movel(pose_trans(ref_frame,p[0.056117, 0.102115, -0.000125, 0.000000, 3.141593, 0.000000]),accel_mss,speed_ms,0,0.001)
    |   movel(pose_trans(ref_frame,p[0.055117, 0.104549, -0.000125, -0.000000, 3.141593, 0.000000]),accel_mss,speed_ms,0,0.001)
    |   movel(pose_trans(ref_frame,p[0.054994, 0.106976, -0.000125, -0.000000, 3.141593, -0.000000]),accel_mss,speed_ms,0,0.001)
    |   movel(pose_trans(ref_frame,p[0.054089, 0.104072, -0.000125, -0.000000, 3.141593, -0.000000]),accel_mss,speed_ms,0,0.001)
    |   movel(pose_trans(ref_frame,p[0.053416, 0.101119, -0.000125, 0.000000, 3.141593, -0.000000]),accel_mss,speed_ms,0,0.001)
    |   movel(pose_trans(ref_frame,p[0.052834, 0.097793, -0.000125, -0.000000, 3.141593, -0.000000]),accel_mss,speed_ms,0,0.001)
    |   movel(pose_trans(ref_frame,p[0.052414, 0.094442, -0.000125, 0.000000, 3.141593, -0.000000]),accel_mss,speed_ms,0,0.001)
    |   movel(pose_trans(ref_frame,p[0.052122, 0.091150, -0.000125, -0.000000, 3.141593, -0.000000]),accel_mss,speed_ms,0,0.001)
    |   movel(pose_trans(ref_frame,p[0.052084, 0.087843, -0.000125, 0.000000, 3.141593, 0.000000]),accel_mss,speed_ms,0,0.001)
    |   movel(pose_trans(ref_frame,p[0.052355, 0.085273, -0.000125, -0.000000, 3.141593, -0.000000]),accel_mss,speed_ms,0,0.001)
    |   movel(pose_trans(ref_frame,p[0.052616, 0.082645, -0.000125, 0.000000, 3.141593, 0.000000]),accel_mss,speed_ms,0,0.001)
    |   movel(pose_trans(ref_frame,p[0.052535, 0.081947, -0.000125, -0.000000, 3.141593, 0.000000]),accel_mss,speed_ms,0,0.001)
    |   movel(pose_trans(ref_frame,p[0.052090, 0.081554, -0.000125, 0.000000, 3.141593, -0.000000]),accel_mss,speed_ms,0,0.001)
    |   movel(pose_trans(ref_frame,p[0.051868, 0.081568, -0.000125, -0.000000, 3.141593, -0.000000]),accel_mss,speed_ms,0,0.001)
    |   movel(pose_trans(ref_frame,p[0.051653, 0.081638, -0.000125, -0.000000, 3.141593, -0.000000]),accel_mss,speed_ms,0,0.001)
    |   movel(pose_trans(ref_frame,p[0.044813, 0.088250, -0.000125, 0.000000, 3.141593, 0.000000]),accel_mss,speed_ms,0,0.001)
    |   movel(pose_trans(ref_frame,p[0.041449, 0.096978, -0.000125, -0.000000, 3.141593, 0.000000]),accel_mss,speed_ms,0,0.001)
    |   movel(pose_trans(ref_frame,p[0.041171, 0.097676, -0.000125, 0.000000, 3.141593, -0.000000]),accel_mss,speed_ms,0,0.001)
    |   movel(pose_trans(ref_frame,p[0.040734, 0.098269, -0.000125, 0.000000, 3.141593, 0.000000]),accel_mss,speed_ms,0,0.001)
    |   movel(pose_trans(ref_frame,p[0.038679, 0.098423, -0.000125, 0.000000, 3.141593, 0.000000]),accel_mss,speed_ms,0,0.001)
    |   movel(pose_trans(ref_frame,p[0.037369, 0.097061, -0.000125, -0.000000, 3.141593, 0.000000]),accel_mss,speed_ms,0,0.001)
    |   movel(pose_trans(ref_frame,p[0.036035, 0.094122, -0.000125, 0.000000, 3.141593, -0.000000]),accel_mss,speed_ms,0,0.001)
    |   movel(pose_trans(ref_frame,p[0.035297, 0.090976, -0.000125, 0.000000, 3.141593, 0.000000]),accel_mss,speed_ms,0,0.001)
    |   movel(pose_trans(ref_frame,p[0.035073, 0.089838, -0.000125, -0.000000, 3.141593, 0.000000]),accel_mss,speed_ms,0,0.001)
    |   movel(pose_trans(ref_frame,p[0.034332, 0.088884, -0.000125, 0.000000, 3.141593, 0.000000]),accel_mss,speed_ms,0,0.001)
    |   movel(pose_trans(ref_frame,p[0.033478, 0.088790, -0.000125, -0.000000, 3.141593, 0.000000]),accel_mss,speed_ms,0,0.001)
    |   movel(pose_trans(ref_frame,p[0.032671, 0.089210, -0.000125, 0.000000, 3.141593, 0.000000]),accel_mss,speed_ms,0,0.001)
    |   movel(pose_trans(ref_frame,p[0.031591, 0.090296, -0.000125, -0.000000, 3.141593, -0.000000]),accel_mss,speed_ms,0,0.001)
    |   movel(pose_trans(ref_frame,p[0.030677, 0.091522, -0.000125, 0.000000, 3.141593, 0.000000]),accel_mss,speed_ms,0,0.001)
    |   movel(pose_trans(ref_frame,p[0.029076, 0.096690, -0.000125, 0.000000, 3.141593, -0.000000]),accel_mss,speed_ms,0,0.001)
    |   movel(pose_trans(ref_frame,p[0.029868, 0.101986, -0.000125, 0.000000, 3.141593, 0.000000]),accel_mss,speed_ms,0,0.001)
    |   movel(pose_trans(ref_frame,p[0.031346, 0.105758, -0.000125, 0.000000, 3.141593, 0.000000]),accel_mss,speed_ms,0,0.001)
    |   movel(pose_trans(ref_frame,p[0.033747, 0.109039, -0.000125, -0.000000, 3.141593, -0.000000]),accel_mss,speed_ms,0,0.001)
    |   movel(pose_trans(ref_frame,p[0.036020, 0.110818, -0.000125, -0.000000, 3.141593, -0.000000]),accel_mss,speed_ms,0,0.001)
    |   movel(pose_trans(ref_frame,p[0.038929, 0.111276, -0.000125, -0.000000, 3.141593, -0.000000]),accel_mss,speed_ms,0,0.001)
    |   movel(pose_trans(ref_frame,p[0.041535, 0.109044, -0.000125, -0.000000, 3.141593, 0.000000]),accel_mss,speed_ms,0,0.001)
    |   movel(pose_trans(ref_frame,p[0.042762, 0.105959, -0.000125, 0.000000, 3.141593, 0.000000]),accel_mss,speed_ms,0,0.001)
    |   movel(pose_trans(ref_frame,p[0.043328, 0.104611, -0.000125, 0.000000, 3.141593, -0.000000]),accel_mss,speed_ms,0,0.001)
    |   movel(pose_trans(ref_frame,p[0.044464, 0.103624, -0.000125, 0.000000, 3.141593, 0.000000]),accel_mss,speed_ms,0,0.001)
    |   movel(pose_trans(ref_frame,p[0.044178, 0.104207, -0.000125, -0.000000, 3.141593, 0.000000]),accel_mss,speed_ms,0,0.001)
    |   movel(pose_trans(ref_frame,p[0.045734, 0.107913, -0.000125, -0.000000, 3.141593, -0.000000]),accel_mss,speed_ms,0,0.001)
    |   movel(pose_trans(ref_frame,p[0.047715, 0.111798, -0.000125, -0.000000, 3.141593, -0.000000]),accel_mss,speed_ms,0,0.001)
    |   movel(pose_trans(ref_frame,p[0.048146, 0.112505, -0.000125, 0.000000, 3.141593, -0.000000]),accel_mss,speed_ms,0,0.001)
    |   movel(pose_trans(ref_frame,p[0.050447, 0.115705, -0.000125, -0.000000, 3.141593, -0.000000]),accel_mss,speed_ms,0,0.001)
    |   movel(pose_trans(ref_frame,p[0.052920, 0.118790, -0.000125, -0.000000, 3.141593, -0.000000]),accel_mss,speed_ms,0,0.001)
    |   movel(pose_trans(ref_frame,p[0.055404, 0.121521, -0.000125, -0.000000, 3.141593, 0.000000]),accel_mss,speed_ms,0,0.001)
    |   movel(pose_trans(ref_frame,p[0.058393, 0.123580, -0.000125, -0.000000, 3.141593, 0.000000]),accel_mss,speed_ms,0,0.001)
    |   movel(pose_trans(ref_frame,p[0.058302, 0.121953, -0.000125, -0.000000, 3.141593, -0.000000]),accel_mss,speed_ms,0,0.001)
    |   movel(pose_trans(ref_frame,p[0.058332, 0.121467, -0.000125, -0.000000, 3.141593, -0.000000]),accel_mss,speed_ms,0,0.001)
    |   movel(pose_trans(ref_frame,p[0.058594, 0.121121, -0.000125, 0.000000, 3.141593, -0.000000]),accel_mss,speed_ms,0,0.001)
    |   movel(pose_trans(ref_frame,p[0.058956, 0.121095, -0.000125, -0.000000, 3.141593, -0.000000]),accel_mss,speed_ms,0,0.001)
    |   movel(pose_trans(ref_frame,p[0.059323, 0.121228, -0.000125, 0.000000, 3.141593, 0.000000]),accel_mss,speed_ms,0,0.001)
    |   movel(pose_trans(ref_frame,p[0.060345, 0.121460, -0.000125, -0.000000, 3.141593, -0.000000]),accel_mss,speed_ms,0,0.001)
    |   movel(pose_trans(ref_frame,p[0.061388, 0.121359, -0.000125, 0.000000, 3.141593, -0.000000]),accel_mss,speed_ms,0,0.001)
    |   movel(pose_trans(ref_frame,p[0.061473, 0.121332, -0.000125, 0.000000, 3.141593, 0.000000]),accel_mss,speed_ms,0,0.001)
    |   movel(pose_trans(ref_frame,p[0.061545, 0.121284, -0.000125, 0.000000, 3.141593, -0.000000]),accel_mss,speed_ms,0,0.001)
    |   movel(pose_trans(ref_frame,p[0.061575, 0.121024, -0.000125, 0.000000, 3.141593, -0.000000]),accel_mss,speed_ms,0,0.001)
    |   movel(pose_trans(ref_frame,p[0.061474, 0.120721, -0.000125, 0.000000, 3.141593, -0.000000]),accel_mss,speed_ms,0,0.001)
    |   movel(pose_trans(ref_frame,p[0.061582, 0.120424, -0.000125, 0.000000, 3.141593, 0.000000]),accel_mss,speed_ms,0,0.001)
    |   movel(pose_trans(ref_frame,p[0.061883, 0.120274, -0.000125, 0.000000, 3.141593, 0.000000]),accel_mss,speed_ms,0,0.001)
    |   movel(pose_trans(ref_frame,p[0.062212, 0.120291, -0.000125, -0.000000, 3.141593, -0.000000]),accel_mss,speed_ms,0,0.001)
    |   movel(pose_trans(ref_frame,p[0.062533, 0.120391, -0.000125, -0.000000, 3.141593, 0.000000]),accel_mss,speed_ms,0,0.001)
    |   movel(pose_trans(ref_frame,p[0.064505, 0.121106, -0.000125, -0.000000, 3.141593, 0.000000]),accel_mss,speed_ms,0,0.001)
    |   movel(pose_trans(ref_frame,p[0.061922, 0.119266, -0.000125, 0.000000, 3.141593, -0.000000]),accel_mss,speed_ms,0,0.001)
    |   movel(pose_trans(ref_frame,p[0.059801, 0.116874, -0.000125, -0.000000, 3.141593, -0.000000]),accel_mss,speed_ms,0,0.001)
    |   movel(pose_trans(ref_frame,p[0.057879, 0.114087, -0.000125, -0.000000, 3.141593, 0.000000]),accel_mss,speed_ms,0,0.001)
    |   movel(pose_trans(ref_frame,p[0.056438, 0.111016, -0.000125, -0.000000, 3.141593, -0.000000]),accel_mss,speed_ms,0,0.001)
    |   movel(pose_trans(ref_frame,p[0.056309, 0.106637, -0.000125, 0.000000, 3.141593, 0.000000]),accel_mss,speed_ms,0,0.001)
    |   movel(pose_trans(ref_frame,p[0.058011, 0.102615, -0.000125, 0.000000, 3.141593, -0.000000]),accel_mss,speed_ms,0,0.001)
    |   movel(pose_trans(ref_frame,p[0.059784, 0.101649, -0.000125, -0.000000, 3.141593, -0.000000]),accel_mss,speed_ms,0,0.001)
    |   movel(pose_trans(ref_frame,p[0.061498, 0.102733, -0.000125, 0.000000, 3.141593, -0.000000]),accel_mss,speed_ms,0,0.001)
    |   movel(pose_trans(ref_frame,p[0.063515, 0.105687, -0.000125, -0.000000, 3.141593, 0.000000]),accel_mss,speed_ms,0,0.001)
    |   movel(pose_trans(ref_frame,p[0.066545, 0.107663, -0.000125, -0.000000, 3.141593, -0.000000]),accel_mss,speed_ms,0,0.001)
    |   movel(pose_trans(ref_frame,p[0.067506, 0.107818, -0.000125, -0.000000, 3.141593, -0.000000]),accel_mss,speed_ms,0,0.001)
    |   movel(pose_trans(ref_frame,p[0.068490, 0.107788, -0.000125, 0.000000, 3.141593, -0.000000]),accel_mss,speed_ms,0,0.001)
    |   movel(pose_trans(ref_frame,p[0.073823, 0.104642, -0.000125, -0.000000, 3.141593, 0.000000]),accel_mss,speed_ms,0,0.001)
    |   movel(pose_trans(ref_frame,p[0.076606, 0.099224, -0.000125, -0.000000, 3.141593, 0.000000]),accel_mss,speed_ms,0,0.001)
    |   movel(pose_trans(ref_frame,p[0.078349, 0.090265, -0.000125, 0.000000, 3.141593, 0.000000]),accel_mss,speed_ms,0,0.001)
    |   movel(pose_trans(ref_frame,p[0.074472, 0.081840, -0.000125, 0.000000, 3.141593, 0.000000]),accel_mss,speed_ms,0,0.001)
    |   movel(pose_trans(ref_frame,p[0.074097, 0.081567, -0.000125, -0.000000, 3.141593, 0.000000]),accel_mss,speed_ms,0,0.001)
    |   movel(pose_trans(ref_frame,p[0.073668, 0.081424, -0.000125, 0.000000, 3.141593, 0.000000]),accel_mss,speed_ms,0,0.001)
    |   movel(pose_trans(ref_frame,p[0.073028, 0.081623, -0.000125, 0.000000, 3.141593, 0.000000]),accel_mss,speed_ms,0,0.001)
    |   movel(pose_trans(ref_frame,p[0.072580, 0.082171, -0.000125, -0.000000, 3.141593, -0.000000]),accel_mss,speed_ms,0,0.001)
    |   movel(pose_trans(ref_frame,p[0.072124, 0.083674, -0.000125, 0.000000, 3.141593, -0.000000]),accel_mss,speed_ms,0,0.001)
    |   movel(pose_trans(ref_frame,p[0.071925, 0.085234, -0.000125, -0.000000, 3.141593, 0.000000]),accel_mss,speed_ms,0,0.001)
    |   movel(pose_trans(ref_frame,p[0.071809, 0.085506, -0.000125, 0.000000, 3.141593, 0.000000]),accel_mss,speed_ms,0,0.001)
    |   movel(pose_trans(ref_frame,p[0.071555, 0.085629, -0.000125, 0.000000, 3.141593, 0.000000]),accel_mss,speed_ms,0,0.001)
    |   movel(pose_trans(ref_frame,p[0.071311, 0.085120, -0.000125, -0.000000, 3.141593, -0.000000]),accel_mss,speed_ms,0,0.001)
    |   movel(pose_trans(ref_frame,p[0.071102, 0.084572, -0.000125, -0.000000, 3.141593, -0.000000]),accel_mss,speed_ms,0,0.001)
    |   movel(pose_trans(ref_frame,p[0.070576, 0.089151, -0.000125, 0.000000, 3.141593, -0.000000]),accel_mss,speed_ms,0,0.001)
    |   movel(pose_trans(ref_frame,p[0.069756, 0.093688, -0.000125, -0.000000, 3.141593, 0.000000]),accel_mss,speed_ms,0,0.001)
    |   movel(pose_trans(ref_frame,p[0.069243, 0.095663, -0.000125, 0.000000, 3.141593, -0.000000]),accel_mss,speed_ms,0,0.001)
    |   movel(pose_trans(ref_frame,p[0.068151, 0.097410, -0.000125, -0.000000, 3.141593, -0.000000]),accel_mss,speed_ms,0,0.001)
    |   movel(pose_trans(ref_frame,p[0.065563, 0.098071, -0.000125, 0.000000, 3.141593, -0.000000]),accel_mss,speed_ms,0,0.001)
    |   movel(pose_trans(ref_frame,p[0.063250, 0.096920, -0.000125, -0.000000, 3.141593, -0.000000]),accel_mss,speed_ms,0,0) # end trace
    |   speed_ms    = 1.000
    |   movel(pose_trans(ref_frame,p[0.063250, 0.096920, 0.005000, -0.000000, 3.141593, -0.000000]),accel_mss,speed_ms,0,0.001)
    |   movel(pose_trans(ref_frame,p[0.059449, 0.103780, 0.005000, 0.000000, 3.141593, -0.000000]),accel_mss,speed_ms,0,0) # end trace
    |   speed_ms    = 0.002
    |   movel(pose_trans(ref_frame,p[0.059449, 0.103780, -0.000125, 0.000000, 3.141593, -0.000000]),accel_mss,speed_ms,0,0) # end trace
    |   speed_ms    = 0.007
    |   movel(pose_trans(ref_frame,p[0.059380, 0.106675, -0.000125, -0.000000, 3.141593, 0.000000]),accel_mss,speed_ms,0,0.001)
    |   movel(pose_trans(ref_frame,p[0.060031, 0.109497, -0.000125, 0.000000, 3.141593, 0.000000]),accel_mss,speed_ms,0,0.001)
    |   movel(pose_trans(ref_frame,p[0.059947, 0.108523, -0.000125, 0.000000, 3.141593, -0.000000]),accel_mss,speed_ms,0,0.001)
    |   movel(pose_trans(ref_frame,p[0.060044, 0.107597, -0.000125, 0.000000, 3.141593, 0.000000]),accel_mss,speed_ms,0,0.001)
    |   movel(pose_trans(ref_frame,p[0.060430, 0.107054, -0.000125, -0.000000, 3.141593, -0.000000]),accel_mss,speed_ms,0,0.001)
    |   movel(pose_trans(ref_frame,p[0.061164, 0.107254, -0.000125, 0.000000, 3.141593, -0.000000]),accel_mss,speed_ms,0,0.001)
    |   movel(pose_trans(ref_frame,p[0.061898, 0.109971, -0.000125, -0.000000, 3.141593, 0.000000]),accel_mss,speed_ms,0,0.001)
    |   movel(pose_trans(ref_frame,p[0.063165, 0.112630, -0.000125, -0.000000, 3.141593, -0.000000]),accel_mss,speed_ms,0,0.001)
    |   movel(pose_trans(ref_frame,p[0.062963, 0.111210, -0.000125, 0.000000, 3.141593, -0.000000]),accel_mss,speed_ms,0,0.001)
    |   movel(pose_trans(ref_frame,p[0.064114, 0.110458, -0.000125, 0.000000, 3.141593, -0.000000]),accel_mss,speed_ms,0,0.001)
    |   movel(pose_trans(ref_frame,p[0.065053, 0.111647, -0.000125, -0.000000, 3.141593, 0.000000]),accel_mss,speed_ms,0,0.001)
    |   movel(pose_trans(ref_frame,p[0.066021, 0.112722, -0.000125, 0.000000, 3.141593, -0.000000]),accel_mss,speed_ms,0,0) # end trace
    |   speed_ms    = 1.000
    |   movel(pose_trans(ref_frame,p[0.066021, 0.112722, 0.005000, 0.000000, 3.141593, 0.000000]),accel_mss,speed_ms,0,0.001)
    |   movel(pose_trans(ref_frame,p[0.063840, 0.108129, 0.005000, -0.000000, 3.141593, 0.000000]),accel_mss,speed_ms,0,0) # end trace
    |   speed_ms    = 0.002
    |   movel(pose_trans(ref_frame,p[0.063840, 0.108129, -0.000125, -0.000000, 3.141593, 0.000000]),accel_mss,speed_ms,0,0) # end trace
    |   speed_ms    = 0.007
    |   movel(pose_trans(ref_frame,p[0.064907, 0.109512, -0.000125, 0.000000, 3.141593, 0.000000]),accel_mss,speed_ms,0,0.001)
    |   movel(pose_trans(ref_frame,p[0.065896, 0.110959, -0.000125, -0.000000, 3.141593, 0.000000]),accel_mss,speed_ms,0,0.001)
    |   movel(pose_trans(ref_frame,p[0.067070, 0.112271, -0.000125, 0.000000, 3.141593, 0.000000]),accel_mss,speed_ms,0,0.001)
    |   movel(pose_trans(ref_frame,p[0.068564, 0.113135, -0.000125, -0.000000, 3.141593, 0.000000]),accel_mss,speed_ms,0,0.001)
    |   movel(pose_trans(ref_frame,p[0.067195, 0.112039, -0.000125, -0.000000, 3.141593, -0.000000]),accel_mss,speed_ms,0,0.001)
    |   movel(pose_trans(ref_frame,p[0.068061, 0.110419, -0.000125, -0.000000, 3.141593, 0.000000]),accel_mss,speed_ms,0,0.001)
    |   movel(pose_trans(ref_frame,p[0.068442, 0.110479, -0.000125, 0.000000, 3.141593, 0.000000]),accel_mss,speed_ms,0,0.001)
    |   movel(pose_trans(ref_frame,p[0.068805, 0.110635, -0.000125, 0.000000, 3.141593, -0.000000]),accel_mss,speed_ms,0,0.001)
    |   movel(pose_trans(ref_frame,p[0.071290, 0.111502, -0.000125, -0.000000, 3.141593, 0.000000]),accel_mss,speed_ms,0,0.001)
    |   movel(pose_trans(ref_frame,p[0.073921, 0.110990, -0.000125, 0.000000, 3.141593, 0.000000]),accel_mss,speed_ms,0,0.001)
    |   movel(pose_trans(ref_frame,p[0.072888, 0.111019, -0.000125, -0.000000, 3.141593, 0.000000]),accel_mss,speed_ms,0,0.001)
    |   movel(pose_trans(ref_frame,p[0.072031, 0.110400, -0.000125, -0.000000, 3.141593, -0.000000]),accel_mss,speed_ms,0,0.001)
    |   movel(pose_trans(ref_frame,p[0.072094, 0.109682, -0.000125, -0.000000, 3.141593, 0.000000]),accel_mss,speed_ms,0,0.001)
    |   movel(pose_trans(ref_frame,p[0.072833, 0.109390, -0.000125, 0.000000, 3.141593, 0.000000]),accel_mss,speed_ms,0,0.001)
    |   movel(pose_trans(ref_frame,p[0.075064, 0.108702, -0.000125, -0.000000, 3.141593, -0.000000]),accel_mss,speed_ms,0,0.001)
    |   movel(pose_trans(ref_frame,p[0.076943, 0.107272, -0.000125, -0.000000, 3.141593, -0.000000]),accel_mss,speed_ms,0,0.001)
    |   movel(pose_trans(ref_frame,p[0.076310, 0.107481, -0.000125, 0.000000, 3.141593, -0.000000]),accel_mss,speed_ms,0,0.001)
    |   movel(pose_trans(ref_frame,p[0.075606, 0.107337, -0.000125, 0.000000, 3.141593, -0.000000]),accel_mss,speed_ms,0,0.001)
    |   movel(pose_trans(ref_frame,p[0.075974, 0.105904, -0.000125, -0.000000, 3.141593, -0.000000]),accel_mss,speed_ms,0,0.001)
    |   movel(pose_trans(ref_frame,p[0.078068, 0.104825, -0.000125, 0.000000, 3.141593, 0.000000]),accel_mss,speed_ms,0,0.001)
    |   movel(pose_trans(ref_frame,p[0.079129, 0.103687, -0.000125, -0.000000, 3.141593, 0.000000]),accel_mss,speed_ms,0,0.001)
    |   movel(pose_trans(ref_frame,p[0.079839, 0.102325, -0.000125, 0.000000, 3.141593, -0.000000]),accel_mss,speed_ms,0,0.001)
    |   movel(pose_trans(ref_frame,p[0.079361, 0.102884, -0.000125, 0.000000, 3.141593, -0.000000]),accel_mss,speed_ms,0,0.001)
    |   movel(pose_trans(ref_frame,p[0.078697, 0.103214, -0.000125, -0.000000, 3.141593, 0.000000]),accel_mss,speed_ms,0,0.001)
    |   movel(pose_trans(ref_frame,p[0.078265, 0.102978, -0.000125, -0.000000, 3.141593, -0.000000]),accel_mss,speed_ms,0,0.001)
    |   movel(pose_trans(ref_frame,p[0.078248, 0.102478, -0.000125, 0.000000, 3.141593, -0.000000]),accel_mss,speed_ms,0,0.001)
    |   movel(pose_trans(ref_frame,p[0.079358, 0.099460, -0.000125, 0.000000, 3.141593, -0.000000]),accel_mss,speed_ms,0,0.001)
    |   movel(pose_trans(ref_frame,p[0.079740, 0.096188, -0.000125, -0.000000, 3.141593, -0.000000]),accel_mss,speed_ms,0,0) # end trace
    |   speed_ms    = 1.000
    |   movel(pose_trans(ref_frame,p[0.079740, 0.096188, 0.005000, -0.000000, 3.141593, 0.000000]),accel_mss,speed_ms,0,0.001)
    |   movel(pose_trans(ref_frame,p[0.069434, 0.088428, 0.005000, -0.000000, 3.141593, -0.000000]),accel_mss,speed_ms,0,0) # end trace
    |   speed_ms    = 0.002
    |   movel(pose_trans(ref_frame,p[0.069434, 0.088428, -0.000125, -0.000000, 3.141593, 0.000000]),accel_mss,speed_ms,0,0) # end trace
    |   speed_ms    = 0.007
    |   movel(pose_trans(ref_frame,p[0.068644, 0.086784, -0.000125, 0.000000, 3.141593, 0.000000]),accel_mss,speed_ms,0,0.001)
    |   movel(pose_trans(ref_frame,p[0.066902, 0.086088, -0.000125, 0.000000, 3.141593, -0.000000]),accel_mss,speed_ms,0,0.001)
    |   movel(pose_trans(ref_frame,p[0.064540, 0.087037, -0.000125, 0.000000, 3.141593, -0.000000]),accel_mss,speed_ms,0,0.001)
    |   movel(pose_trans(ref_frame,p[0.063232, 0.089163, -0.000125, -0.000000, 3.141593, 0.000000]),accel_mss,speed_ms,0,0.001)
    |   movel(pose_trans(ref_frame,p[0.063410, 0.093674, -0.000125, -0.000000, 3.141593, -0.000000]),accel_mss,speed_ms,0,0.001)
    |   movel(pose_trans(ref_frame,p[0.066314, 0.097161, -0.000125, -0.000000, 3.141593, 0.000000]),accel_mss,speed_ms,0,0) # end trace
    |   speed_ms    = 1.000
    |   movel(pose_trans(ref_frame,p[0.066314, 0.097161, 0.005000, -0.000000, 3.141593, -0.000000]),accel_mss,speed_ms,0,0.001)
    |   movel(pose_trans(ref_frame,p[0.043879, 0.107183, 0.005000, 0.000000, 3.141593, 0.000000]),accel_mss,speed_ms,0,0) # end trace
    |   speed_ms    = 0.002
    |   movel(pose_trans(ref_frame,p[0.043879, 0.107183, -0.000125, 0.000000, 3.141593, 0.000000]),accel_mss,speed_ms,0,0) # end trace
    |   speed_ms    = 0.007
    |   movel(pose_trans(ref_frame,p[0.043949, 0.109689, -0.000125, 0.000000, 3.141593, 0.000000]),accel_mss,speed_ms,0,0.001)
    |   movel(pose_trans(ref_frame,p[0.044358, 0.112191, -0.000125, 0.000000, 3.141593, -0.000000]),accel_mss,speed_ms,0,0.001)
    |   movel(pose_trans(ref_frame,p[0.044600, 0.112830, -0.000125, -0.000000, 3.141593, 0.000000]),accel_mss,speed_ms,0,0.001)
    |   movel(pose_trans(ref_frame,p[0.044974, 0.113392, -0.000125, 0.000000, 3.141593, 0.000000]),accel_mss,speed_ms,0,0.001)
    |   movel(pose_trans(ref_frame,p[0.045047, 0.112783, -0.000125, -0.000000, 3.141593, -0.000000]),accel_mss,speed_ms,0,0.001)
    |   movel(pose_trans(ref_frame,p[0.045212, 0.112191, -0.000125, -0.000000, 3.141593, -0.000000]),accel_mss,speed_ms,0,0.001)
    |   movel(pose_trans(ref_frame,p[0.045255, 0.112092, -0.000125, -0.000000, 3.141593, -0.000000]),accel_mss,speed_ms,0,0.001)
    |   movel(pose_trans(ref_frame,p[0.045321, 0.112013, -0.000125, -0.000000, 3.141593, -0.000000]),accel_mss,speed_ms,0,0.001)
    |   movel(pose_trans(ref_frame,p[0.045524, 0.111982, -0.000125, -0.000000, 3.141593, 0.000000]),accel_mss,speed_ms,0,0.001)
    |   movel(pose_trans(ref_frame,p[0.045725, 0.112094, -0.000125, -0.000000, 3.141593, -0.000000]),accel_mss,speed_ms,0,0.001)
    |   movel(pose_trans(ref_frame,p[0.046450, 0.113364, -0.000125, 0.000000, 3.141593, -0.000000]),accel_mss,speed_ms,0,0.001)
    |   movel(pose_trans(ref_frame,p[0.046706, 0.114775, -0.000125, 0.000000, 3.141593, -0.000000]),accel_mss,speed_ms,0,0.001)
    |   movel(pose_trans(ref_frame,p[0.047171, 0.116428, -0.000125, 0.000000, 3.141593, -0.000000]),accel_mss,speed_ms,0,0.001)
    |   movel(pose_trans(ref_frame,p[0.047952, 0.117961, -0.000125, 0.000000, 3.141593, 0.000000]),accel_mss,speed_ms,0,0.001)
    |   movel(pose_trans(ref_frame,p[0.047879, 0.117282, -0.000125, -0.000000, 3.141593, 0.000000]),accel_mss,speed_ms,0,0.001)
    |   movel(pose_trans(ref_frame,p[0.047964, 0.116605, -0.000125, 0.000000, 3.141593, 0.000000]),accel_mss,speed_ms,0,0.001)
    |   movel(pose_trans(ref_frame,p[0.048020, 0.116440, -0.000125, -0.000000, 3.141593, 0.000000]),accel_mss,speed_ms,0,0.001)
    |   movel(pose_trans(ref_frame,p[0.048129, 0.116311, -0.000125, -0.000000, 3.141593, 0.000000]),accel_mss,speed_ms,0,0.001)
    |   movel(pose_trans(ref_frame,p[0.048393, 0.116283, -0.000125, 0.000000, 3.141593, 0.000000]),accel_mss,speed_ms,0,0.001)
    |   movel(pose_trans(ref_frame,p[0.048646, 0.116433, -0.000125, -0.000000, 3.141593, -0.000000]),accel_mss,speed_ms,0,0.001)
    |   movel(pose_trans(ref_frame,p[0.049455, 0.117693, -0.000125, 0.000000, 3.141593, -0.000000]),accel_mss,speed_ms,0,0.001)
    |   movel(pose_trans(ref_frame,p[0.049946, 0.119102, -0.000125, -0.000000, 3.141593, -0.000000]),accel_mss,speed_ms,0,0.001)
    |   movel(pose_trans(ref_frame,p[0.050710, 0.120593, -0.000125, -0.000000, 3.141593, 0.000000]),accel_mss,speed_ms,0,0.001)
    |   movel(pose_trans(ref_frame,p[0.051783, 0.121885, -0.000125, 0.000000, 3.141593, 0.000000]),accel_mss,speed_ms,0,0.001)
    |   movel(pose_trans(ref_frame,p[0.051644, 0.121153, -0.000125, 0.000000, 3.141593, -0.000000]),accel_mss,speed_ms,0,0.001)
    |   movel(pose_trans(ref_frame,p[0.051689, 0.120409, -0.000125, -0.000000, 3.141593, -0.000000]),accel_mss,speed_ms,0,0.001)
    |   movel(pose_trans(ref_frame,p[0.051746, 0.120242, -0.000125, 0.000000, 3.141593, 0.000000]),accel_mss,speed_ms,0,0.001)
    |   movel(pose_trans(ref_frame,p[0.051874, 0.120153, -0.000125, 0.000000, 3.141593, -0.000000]),accel_mss,speed_ms,0,0.001)
    |   movel(pose_trans(ref_frame,p[0.051959, 0.120167, -0.000125, 0.000000, 3.141593, 0.000000]),accel_mss,speed_ms,0,0.001)
    |   movel(pose_trans(ref_frame,p[0.052037, 0.120208, -0.000125, -0.000000, 3.141593, 0.000000]),accel_mss,speed_ms,0,0.001)
    |   movel(pose_trans(ref_frame,p[0.053197, 0.121434, -0.000125, -0.000000, 3.141593, 0.000000]),accel_mss,speed_ms,0,0.001)
    |   movel(pose_trans(ref_frame,p[0.054263, 0.122745, -0.000125, -0.000000, 3.141593, -0.000000]),accel_mss,speed_ms,0,0.001)
    |   movel(pose_trans(ref_frame,p[0.055986, 0.123997, -0.000125, -0.000000, 3.141593, -0.000000]),accel_mss,speed_ms,0,0.001)
    |   movel(pose_trans(ref_frame,p[0.057836, 0.125048, -0.000125, 0.000000, 3.141593, 0.000000]),accel_mss,speed_ms,0,0) # end trace
    |   speed_ms    = 1.000
    |   movel(pose_trans(ref_frame,p[0.057836, 0.125048, 0.005000, 0.000000, 3.141593, 0.000000]),accel_mss,speed_ms,0,0.001)
    |   movel(pose_trans(ref_frame,p[0.042652, 0.078559, 0.005000, -0.000000, 3.141593, 0.000000]),accel_mss,speed_ms,0,0) # end trace
    |   speed_ms    = 0.002
    |   movel(pose_trans(ref_frame,p[0.042652, 0.078559, -0.000125, -0.000000, 3.141593, 0.000000]),accel_mss,speed_ms,0,0) # end trace
    |   speed_ms    = 0.007
    |   movel(pose_trans(ref_frame,p[0.045257, 0.077566, -0.000125, 0.000000, 3.141593, 0.000000]),accel_mss,speed_ms,0,0.001)
    |   movel(pose_trans(ref_frame,p[0.047013, 0.075414, -0.000125, -0.000000, 3.141593, 0.000000]),accel_mss,speed_ms,0,0.001)
    |   movel(pose_trans(ref_frame,p[0.046026, 0.075734, -0.000125, -0.000000, 3.141593, -0.000000]),accel_mss,speed_ms,0,0.001)
    |   movel(pose_trans(ref_frame,p[0.044988, 0.075834, -0.000125, 0.000000, 3.141593, -0.000000]),accel_mss,speed_ms,0,0.001)
    |   movel(pose_trans(ref_frame,p[0.044598, 0.075766, -0.000125, 0.000000, 3.141593, 0.000000]),accel_mss,speed_ms,0,0.001)
    |   movel(pose_trans(ref_frame,p[0.044339, 0.075518, -0.000125, 0.000000, 3.141593, 0.000000]),accel_mss,speed_ms,0,0.001)
    |   movel(pose_trans(ref_frame,p[0.044401, 0.075113, -0.000125, -0.000000, 3.141593, -0.000000]),accel_mss,speed_ms,0,0.001)
    |   movel(pose_trans(ref_frame,p[0.044731, 0.074783, -0.000125, -0.000000, 3.141593, 0.000000]),accel_mss,speed_ms,0,0.001)
    |   movel(pose_trans(ref_frame,p[0.045965, 0.073787, -0.000125, 0.000000, 3.141593, 0.000000]),accel_mss,speed_ms,0,0.001)
    |   movel(pose_trans(ref_frame,p[0.047037, 0.072608, -0.000125, -0.000000, 3.141593, -0.000000]),accel_mss,speed_ms,0,0.001)
    |   movel(pose_trans(ref_frame,p[0.047851, 0.071217, -0.000125, 0.000000, 3.141593, 0.000000]),accel_mss,speed_ms,0,0.001)
    |   movel(pose_trans(ref_frame,p[0.048462, 0.069725, -0.000125, 0.000000, 3.141593, -0.000000]),accel_mss,speed_ms,0,0.001)
    |   movel(pose_trans(ref_frame,p[0.047975, 0.069944, -0.000125, 0.000000, 3.141593, 0.000000]),accel_mss,speed_ms,0,0.001)
    |   movel(pose_trans(ref_frame,p[0.047465, 0.070071, -0.000125, -0.000000, 3.141593, -0.000000]),accel_mss,speed_ms,0,0.001)
    |   movel(pose_trans(ref_frame,p[0.047172, 0.069997, -0.000125, 0.000000, 3.141593, -0.000000]),accel_mss,speed_ms,0,0.001)
    |   movel(pose_trans(ref_frame,p[0.046995, 0.069770, -0.000125, -0.000000, 3.141593, 0.000000]),accel_mss,speed_ms,0,0.001)
    |   movel(pose_trans(ref_frame,p[0.047514, 0.068756, -0.000125, 0.000000, 3.141593, -0.000000]),accel_mss,speed_ms,0,0.001)
    |   movel(pose_trans(ref_frame,p[0.049186, 0.067485, -0.000125, -0.000000, 3.141593, 0.000000]),accel_mss,speed_ms,0,0.001)
    |   movel(pose_trans(ref_frame,p[0.050078, 0.065924, -0.000125, -0.000000, 3.141593, 0.000000]),accel_mss,speed_ms,0,0.001)
    |   movel(pose_trans(ref_frame,p[0.050444, 0.064923, -0.000125, 0.000000, 3.141593, -0.000000]),accel_mss,speed_ms,0,0.001)
    |   movel(pose_trans(ref_frame,p[0.049565, 0.065365, -0.000125, 0.000000, 3.141593, 0.000000]),accel_mss,speed_ms,0,0.001)
    |   movel(pose_trans(ref_frame,p[0.048678, 0.065094, -0.000125, 0.000000, 3.141593, 0.000000]),accel_mss,speed_ms,0,0.001)
    |   movel(pose_trans(ref_frame,p[0.048662, 0.064951, -0.000125, 0.000000, 3.141593, -0.000000]),accel_mss,speed_ms,0,0.001)
    |   movel(pose_trans(ref_frame,p[0.048701, 0.064806, -0.000125, 0.000000, 3.141593, -0.000000]),accel_mss,speed_ms,0,0.001)
    |   movel(pose_trans(ref_frame,p[0.049407, 0.063515, -0.000125, 0.000000, 3.141593, 0.000000]),accel_mss,speed_ms,0,0.001)
    |   movel(pose_trans(ref_frame,p[0.050149, 0.062182, -0.000125, -0.000000, 3.141593, -0.000000]),accel_mss,speed_ms,0,0.001)
    |   movel(pose_trans(ref_frame,p[0.050518, 0.060477, -0.000125, -0.000000, 3.141593, -0.000000]),accel_mss,speed_ms,0,0.001)
    |   movel(pose_trans(ref_frame,p[0.050630, 0.058731, -0.000125, -0.000000, 3.141593, 0.000000]),accel_mss,speed_ms,0,0.001)
    |   movel(pose_trans(ref_frame,p[0.049919, 0.060522, -0.000125, -0.000000, 3.141593, -0.000000]),accel_mss,speed_ms,0,0.001)
    |   movel(pose_trans(ref_frame,p[0.048568, 0.061760, -0.000125, 0.000000, 3.141593, 0.000000]),accel_mss,speed_ms,0,0.001)
    |   movel(pose_trans(ref_frame,p[0.048480, 0.061793, -0.000125, -0.000000, 3.141593, -0.000000]),accel_mss,speed_ms,0,0.001)
    |   movel(pose_trans(ref_frame,p[0.048388, 0.061800, -0.000125, 0.000000, 3.141593, 0.000000]),accel_mss,speed_ms,0,0.001)
    |   movel(pose_trans(ref_frame,p[0.048204, 0.061586, -0.000125, 0.000000, 3.141593, -0.000000]),accel_mss,speed_ms,0,0.001)
    |   movel(pose_trans(ref_frame,p[0.048282, 0.061224, -0.000125, -0.000000, 3.141593, 0.000000]),accel_mss,speed_ms,0,0.001)
    |   movel(pose_trans(ref_frame,p[0.049556, 0.057639, -0.000125, 0.000000, 3.141593, 0.000000]),accel_mss,speed_ms,0,0.001)
    |   movel(pose_trans(ref_frame,p[0.049582, 0.053825, -0.000125, 0.000000, 3.141593, -0.000000]),accel_mss,speed_ms,0,0.001)
    |   movel(pose_trans(ref_frame,p[0.049624, 0.055908, -0.000125, 0.000000, 3.141593, -0.000000]),accel_mss,speed_ms,0,0.001)
    |   movel(pose_trans(ref_frame,p[0.047652, 0.056705, -0.000125, 0.000000, 3.141593, 0.000000]),accel_mss,speed_ms,0,0.001)
    |   movel(pose_trans(ref_frame,p[0.047606, 0.056590, -0.000125, -0.000000, 3.141593, 0.000000]),accel_mss,speed_ms,0,0.001)
    |   movel(pose_trans(ref_frame,p[0.047594, 0.056465, -0.000125, 0.000000, 3.141593, 0.000000]),accel_mss,speed_ms,0,0.001)
    |   movel(pose_trans(ref_frame,p[0.048432, 0.053555, -0.000125, 0.000000, 3.141593, -0.000000]),accel_mss,speed_ms,0,0.001)
    |   movel(pose_trans(ref_frame,p[0.048123, 0.050736, -0.000125, 0.000000, 3.141593, -0.000000]),accel_mss,speed_ms,0,0) # end trace
    |   speed_ms    = 1.000
    |   movel(pose_trans(ref_frame,p[0.048123, 0.050736, 0.005000, 0.000000, 3.141593, 0.000000]),accel_mss,speed_ms,0,0.001)
    |   movel(pose_trans(ref_frame,p[0.038483, 0.046314, 0.005000, -0.000000, 3.141593, 0.000000]),accel_mss,speed_ms,0,0) # end trace
    |   speed_ms    = 0.002
    |   movel(pose_trans(ref_frame,p[0.038483, 0.046314, -0.000125, -0.000000, 3.141593, -0.000000]),accel_mss,speed_ms,0,0) # end trace
    |   speed_ms    = 0.007
    |   movel(pose_trans(ref_frame,p[0.039565, 0.043108, -0.000125, -0.000000, 3.141593, -0.000000]),accel_mss,speed_ms,0,0.001)
    |   movel(pose_trans(ref_frame,p[0.042032, 0.040715, -0.000125, -0.000000, 3.141593, -0.000000]),accel_mss,speed_ms,0,0) # end trace
    |   speed_ms    = 1.000
    |   movel(pose_trans(ref_frame,p[0.042032, 0.040715, 0.005000, -0.000000, 3.141593, -0.000000]),accel_mss,speed_ms,0,0.001)
    |   movel(pose_trans(ref_frame,p[0.038688, 0.041504, 0.005000, -0.000000, 3.141593, -0.000000]),accel_mss,speed_ms,0,0) # end trace
    |   speed_ms    = 0.002
    |   movel(pose_trans(ref_frame,p[0.038688, 0.041504, -0.000125, -0.000000, 3.141593, 0.000000]),accel_mss,speed_ms,0,0) # end trace
    |   speed_ms    = 0.007
    |   movel(pose_trans(ref_frame,p[0.039258, 0.037487, -0.000125, -0.000000, 3.141593, 0.000000]),accel_mss,speed_ms,0,0.001)
    |   movel(pose_trans(ref_frame,p[0.041760, 0.034196, -0.000125, 0.000000, 3.141593, 0.000000]),accel_mss,speed_ms,0,0) # end trace
    |   speed_ms    = 1.000
    |   movel(pose_trans(ref_frame,p[0.041760, 0.034196, 0.005000, -0.000000, 3.141593, 0.000000]),accel_mss,speed_ms,0,0.001)
    |   movel(pose_trans(ref_frame,p[0.038321, 0.034883, 0.005000, -0.000000, 3.141593, 0.000000]),accel_mss,speed_ms,0,0) # end trace
    |   speed_ms    = 0.002
    |   movel(pose_trans(ref_frame,p[0.038321, 0.034883, -0.000125, -0.000000, 3.141593, 0.000000]),accel_mss,speed_ms,0,0) # end trace
    |   speed_ms    = 0.007
    |   movel(pose_trans(ref_frame,p[0.038895, 0.030356, -0.000125, -0.000000, 3.141593, 0.000000]),accel_mss,speed_ms,0,0.001)
    |   movel(pose_trans(ref_frame,p[0.041911, 0.026822, -0.000125, -0.000000, 3.141593, -0.000000]),accel_mss,speed_ms,0,0) # end trace
    |   speed_ms    = 1.000
    |   movel(pose_trans(ref_frame,p[0.041911, 0.026822, 0.005000, -0.000000, 3.141593, -0.000000]),accel_mss,speed_ms,0,0.001)
    |   movel(pose_trans(ref_frame,p[0.037829, 0.027381, 0.005000, -0.000000, 3.141593, -0.000000]),accel_mss,speed_ms,0,0) # end trace
    |   speed_ms    = 0.002
    |   movel(pose_trans(ref_frame,p[0.037829, 0.027381, -0.000125, -0.000000, 3.141593, -0.000000]),accel_mss,speed_ms,0,0) # end trace
    |   speed_ms    = 0.007
    |   movel(pose_trans(ref_frame,p[0.037791, 0.027489, -0.000125, -0.000000, 3.141593, 0.000000]),accel_mss,speed_ms,0,0.001)
    |   movel(pose_trans(ref_frame,p[0.037753, 0.027596, -0.000125, -0.000000, 3.141593, 0.000000]),accel_mss,speed_ms,0,0.001)
    |   movel(pose_trans(ref_frame,p[0.038872, 0.022718, -0.000125, -0.000000, 3.141593, -0.000000]),accel_mss,speed_ms,0,0.001)
    |   movel(pose_trans(ref_frame,p[0.043044, 0.019776, -0.000125, 0.000000, 3.141593, -0.000000]),accel_mss,speed_ms,0,0) # end trace
    |   speed_ms    = 1.000
    |   movel(pose_trans(ref_frame,p[0.043044, 0.019776, 0.005000, 0.000000, 3.141593, 0.000000]),accel_mss,speed_ms,0,0.001)
    |   movel(pose_trans(ref_frame,p[0.038191, 0.020384, 0.005000, 0.000000, 3.141593, -0.000000]),accel_mss,speed_ms,0,0) # end trace
    |   speed_ms    = 0.002
    |   movel(pose_trans(ref_frame,p[0.038191, 0.020384, -0.000125, 0.000000, 3.141593, -0.000000]),accel_mss,speed_ms,0,0) # end trace
    |   speed_ms    = 0.007
    |   movel(pose_trans(ref_frame,p[0.038588, 0.017563, -0.000125, -0.000000, 3.141593, -0.000000]),accel_mss,speed_ms,0,0.001)
    |   movel(pose_trans(ref_frame,p[0.040507, 0.015396, -0.000125, -0.000000, 3.141593, -0.000000]),accel_mss,speed_ms,0,0.001)
    |   movel(pose_trans(ref_frame,p[0.043138, 0.014744, -0.000125, -0.000000, 3.141593, 0.000000]),accel_mss,speed_ms,0,0.001)
    |   movel(pose_trans(ref_frame,p[0.045763, 0.015491, -0.000125, -0.000000, 3.141593, 0.000000]),accel_mss,speed_ms,0,0) # end trace
    |   speed_ms    = 1.000
    |   movel(pose_trans(ref_frame,p[0.045763, 0.015491, 0.005000, -0.000000, 3.141593, -0.000000]),accel_mss,speed_ms,0,0.001)
    |   movel(pose_trans(ref_frame,p[0.040024, 0.012488, 0.005000, 0.000000, 3.141593, -0.000000]),accel_mss,speed_ms,0,0) # end trace
    |   speed_ms    = 0.002
    |   movel(pose_trans(ref_frame,p[0.040024, 0.012488, -0.000125, 0.000000, 3.141593, 0.000000]),accel_mss,speed_ms,0,0) # end trace
    |   speed_ms    = 0.007
    |   movel(pose_trans(ref_frame,p[0.042423, 0.009833, -0.000125, 0.000000, 3.141593, 0.000000]),accel_mss,speed_ms,0,0.001)
    |   movel(pose_trans(ref_frame,p[0.045846, 0.008791, -0.000125, -0.000000, 3.141593, -0.000000]),accel_mss,speed_ms,0,0.001)
    |   movel(pose_trans(ref_frame,p[0.049298, 0.009684, -0.000125, 0.000000, 3.141593, -0.000000]),accel_mss,speed_ms,0,0.001)
    |   movel(pose_trans(ref_frame,p[0.051149, 0.012821, -0.000125, 0.000000, 3.141593, -0.000000]),accel_mss,speed_ms,0,0) # end trace
    |   speed_ms    = 1.000
    |   movel(pose_trans(ref_frame,p[0.051149, 0.012821, 0.005000, 0.000000, 3.141593, -0.000000]),accel_mss,speed_ms,0,0.001)
    |   movel(pose_trans(ref_frame,p[0.053984, 0.004195, 0.005000, 0.000000, 3.141593, 0.000000]),accel_mss,speed_ms,0,0) # end trace
    |   speed_ms    = 0.002
    |   movel(pose_trans(ref_frame,p[0.053984, 0.004195, -0.000125, 0.000000, 3.141593, -0.000000]),accel_mss,speed_ms,0,0) # end trace
    |   speed_ms    = 0.007
    |   movel(pose_trans(ref_frame,p[0.058130, 0.007905, -0.000125, -0.000000, 3.141593, -0.000000]),accel_mss,speed_ms,0,0.001)
    |   movel(pose_trans(ref_frame,p[0.058089, 0.013936, -0.000125, 0.000000, 3.141593, 0.000000]),accel_mss,speed_ms,0,0) # end trace
    |   speed_ms    = 1.000
    |   movel(pose_trans(ref_frame,p[0.058089, 0.013936, 0.005000, 0.000000, 3.141593, -0.000000]),accel_mss,speed_ms,0,0.001)
    |   movel(pose_trans(ref_frame,p[0.059942, 0.009963, 0.005000, 0.000000, 3.141593, -0.000000]),accel_mss,speed_ms,0,0) # end trace
    |   speed_ms    = 0.002
    |   movel(pose_trans(ref_frame,p[0.059942, 0.009963, -0.000125, 0.000000, 3.141593, 0.000000]),accel_mss,speed_ms,0,0) # end trace
    |   speed_ms    = 0.007
    |   movel(pose_trans(ref_frame,p[0.061336, 0.013374, -0.000125, 0.000000, 3.141593, -0.000000]),accel_mss,speed_ms,0,0.001)
    |   movel(pose_trans(ref_frame,p[0.060818, 0.017101, -0.000125, 0.000000, 3.141593, -0.000000]),accel_mss,speed_ms,0,0) # end trace
    |   speed_ms    = 1.000
    |   movel(pose_trans(ref_frame,p[0.060818, 0.017101, 0.005000, 0.000000, 3.141593, -0.000000]),accel_mss,speed_ms,0,0.001)
    |   movel(pose_trans(ref_frame,p[0.062327, 0.016362, 0.005000, -0.000000, 3.141593, -0.000000]),accel_mss,speed_ms,0,0) # end trace
    |   speed_ms    = 0.002
    |   movel(pose_trans(ref_frame,p[0.062327, 0.016362, -0.000125, -0.000000, 3.141593, 0.000000]),accel_mss,speed_ms,0,0) # end trace
    |   speed_ms    = 0.007
    |   movel(pose_trans(ref_frame,p[0.062617, 0.018444, -0.000125, 0.000000, 3.141593, -0.000000]),accel_mss,speed_ms,0,0.001)
    |   movel(pose_trans(ref_frame,p[0.062408, 0.020546, -0.000125, -0.000000, 3.141593, -0.000000]),accel_mss,speed_ms,0,0) # end trace
    |   speed_ms    = 1.000
    |   movel(pose_trans(ref_frame,p[0.062408, 0.020546, 0.005000, -0.000000, 3.141593, -0.000000]),accel_mss,speed_ms,0,0.001)
    |   movel(pose_trans(ref_frame,p[0.062553, 0.023715, 0.005000, 0.000000, 3.141593, -0.000000]),accel_mss,speed_ms,0,0) # end trace
    |   speed_ms    = 0.002
    |   movel(pose_trans(ref_frame,p[0.062553, 0.023715, -0.000125, 0.000000, 3.141593, 0.000000]),accel_mss,speed_ms,0,0) # end trace
    |   speed_ms    = 0.007
    |   movel(pose_trans(ref_frame,p[0.064503, 0.020311, -0.000125, 0.000000, 3.141593, 0.000000]),accel_mss,speed_ms,0,0.001)
    |   movel(pose_trans(ref_frame,p[0.068164, 0.018929, -0.000125, 0.000000, 3.141593, -0.000000]),accel_mss,speed_ms,0,0) # end trace
    |   speed_ms    = 1.000
    |   movel(pose_trans(ref_frame,p[0.068164, 0.018929, 0.005000, 0.000000, 3.141593, 0.000000]),accel_mss,speed_ms,0,0.001)
    |   movel(pose_trans(ref_frame,p[0.065205, 0.017987, 0.005000, 0.000000, 3.141593, 0.000000]),accel_mss,speed_ms,0,0) # end trace
    |   speed_ms    = 0.002
    |   movel(pose_trans(ref_frame,p[0.065205, 0.017987, -0.000125, 0.000000, 3.141593, 0.000000]),accel_mss,speed_ms,0,0) # end trace
    |   speed_ms    = 0.007
    |   movel(pose_trans(ref_frame,p[0.068259, 0.014838, -0.000125, 0.000000, 3.141593, -0.000000]),accel_mss,speed_ms,0,0.001)
    |   movel(pose_trans(ref_frame,p[0.072604, 0.013978, -0.000125, -0.000000, 3.141593, 0.000000]),accel_mss,speed_ms,0,0) # end trace
    |   speed_ms    = 1.000
    |   movel(pose_trans(ref_frame,p[0.072604, 0.013978, 0.005000, -0.000000, 3.141593, -0.000000]),accel_mss,speed_ms,0,0.001)
    |   movel(pose_trans(ref_frame,p[0.069497, 0.012518, 0.005000, -0.000000, 3.141593, 0.000000]),accel_mss,speed_ms,0,0) # end trace
    |   speed_ms    = 0.002
    |   movel(pose_trans(ref_frame,p[0.069497, 0.012518, -0.000125, -0.000000, 3.141593, -0.000000]),accel_mss,speed_ms,0,0) # end trace
    |   speed_ms    = 0.007
    |   movel(pose_trans(ref_frame,p[0.070014, 0.011257, -0.000125, -0.000000, 3.141593, 0.000000]),accel_mss,speed_ms,0,0.001)
    |   movel(pose_trans(ref_frame,p[0.070855, 0.010184, -0.000125, 0.000000, 3.141593, 0.000000]),accel_mss,speed_ms,0,0.001)
    |   movel(pose_trans(ref_frame,p[0.071490, 0.009657, -0.000125, -0.000000, 3.141593, -0.000000]),accel_mss,speed_ms,0,0.001)
    |   movel(pose_trans(ref_frame,p[0.072186, 0.009212, -0.000125, -0.000000, 3.141593, -0.000000]),accel_mss,speed_ms,0,0.001)
    |   movel(pose_trans(ref_frame,p[0.073966, 0.008425, -0.000125, -0.000000, 3.141593, -0.000000]),accel_mss,speed_ms,0,0.001)
    |   movel(pose_trans(ref_frame,p[0.075877, 0.008111, -0.000125, 0.000000, 3.141593, -0.000000]),accel_mss,speed_ms,0,0.001)
    |   movel(pose_trans(ref_frame,p[0.077796, 0.008409, -0.000125, 0.000000, 3.141593, -0.000000]),accel_mss,speed_ms,0,0.001)
    |   movel(pose_trans(ref_frame,p[0.079454, 0.009391, -0.000125, -0.000000, 3.141593, -0.000000]),accel_mss,speed_ms,0,0) # end trace
    |   speed_ms    = 1.000
    |   movel(pose_trans(ref_frame,p[0.079454, 0.009391, 0.005000, -0.000000, 3.141593, -0.000000]),accel_mss,speed_ms,0,0.001)
    |   movel(pose_trans(ref_frame,p[0.076139, 0.006518, 0.005000, -0.000000, 3.141593, -0.000000]),accel_mss,speed_ms,0,0) # end trace
    |   speed_ms    = 0.002
    |   movel(pose_trans(ref_frame,p[0.076139, 0.006518, -0.000125, -0.000000, 3.141593, -0.000000]),accel_mss,speed_ms,0,0) # end trace
    |   speed_ms    = 0.007
    |   movel(pose_trans(ref_frame,p[0.080860, 0.005172, -0.000125, -0.000000, 3.141593, 0.000000]),accel_mss,speed_ms,0,0.001)
    |   movel(pose_trans(ref_frame,p[0.085553, 0.006939, -0.000125, 0.000000, 3.141593, -0.000000]),accel_mss,speed_ms,0,0) # end trace
    |   speed_ms    = 1.000
    |   movel(pose_trans(ref_frame,p[0.085553, 0.006939, 0.005000, 0.000000, 3.141593, -0.000000]),accel_mss,speed_ms,0,0.001)
    |   movel(pose_trans(ref_frame,p[0.083116, 0.003097, 0.005000, 0.000000, 3.141593, -0.000000]),accel_mss,speed_ms,0,0) # end trace
    |   speed_ms    = 0.002
    |   movel(pose_trans(ref_frame,p[0.083116, 0.003097, -0.000125, 0.000000, 3.141593, -0.000000]),accel_mss,speed_ms,0,0) # end trace
    |   speed_ms    = 0.007
    |   movel(pose_trans(ref_frame,p[0.085539, 0.002500, -0.000125, -0.000000, 3.141593, -0.000000]),accel_mss,speed_ms,0,0.001)
    |   movel(pose_trans(ref_frame,p[0.088011, 0.002836, -0.000125, 0.000000, 3.141593, -0.000000]),accel_mss,speed_ms,0,0.001)
    |   movel(pose_trans(ref_frame,p[0.090187, 0.004057, -0.000125, -0.000000, 3.141593, -0.000000]),accel_mss,speed_ms,0,0.001)
    |   movel(pose_trans(ref_frame,p[0.091761, 0.005992, -0.000125, 0.000000, 3.141593, -0.000000]),accel_mss,speed_ms,0,0) # end trace
    |   speed_ms    = 1.000
    |   movel(pose_trans(ref_frame,p[0.091761, 0.005992, 0.005000, 0.000000, 3.141593, -0.000000]),accel_mss,speed_ms,0,0.001)
    |   movel(pose_trans(ref_frame,p[0.090259, 0.001894, 0.005000, 0.000000, 3.141593, -0.000000]),accel_mss,speed_ms,0,0) # end trace
    |   speed_ms    = 0.002
    |   movel(pose_trans(ref_frame,p[0.090259, 0.001894, -0.000125, 0.000000, 3.141593, -0.000000]),accel_mss,speed_ms,0,0) # end trace
    |   speed_ms    = 0.007
    |   movel(pose_trans(ref_frame,p[0.092648, 0.001669, -0.000125, 0.000000, 3.141593, -0.000000]),accel_mss,speed_ms,0,0.001)
    |   movel(pose_trans(ref_frame,p[0.094938, 0.002657, -0.000125, -0.000000, 3.141593, -0.000000]),accel_mss,speed_ms,0,0.001)
    |   movel(pose_trans(ref_frame,p[0.096806, 0.004399, -0.000125, -0.000000, 3.141593, -0.000000]),accel_mss,speed_ms,0,0.001)
    |   movel(pose_trans(ref_frame,p[0.097701, 0.006720, -0.000125, -0.000000, 3.141593, -0.000000]),accel_mss,speed_ms,0,0) # end trace
    |   speed_ms    = 1.000
    |   movel(pose_trans(ref_frame,p[0.097701, 0.006720, 0.005000, -0.000000, 3.141593, 0.000000]),accel_mss,speed_ms,0,0.001)
    |   movel(pose_trans(ref_frame,p[0.097683, 0.002768, 0.005000, 0.000000, 3.141593, -0.000000]),accel_mss,speed_ms,0,0) # end trace
    |   speed_ms    = 0.002
    |   movel(pose_trans(ref_frame,p[0.097683, 0.002768, -0.000125, 0.000000, 3.141593, 0.000000]),accel_mss,speed_ms,0,0) # end trace
    |   speed_ms    = 0.007
    |   movel(pose_trans(ref_frame,p[0.101003, 0.004037, -0.000125, 0.000000, 3.141593, -0.000000]),accel_mss,speed_ms,0,0.001)
    |   movel(pose_trans(ref_frame,p[0.102515, 0.007301, -0.000125, 0.000000, 3.141593, -0.000000]),accel_mss,speed_ms,0,0) # end trace
    |   speed_ms    = 1.000
    |   movel(pose_trans(ref_frame,p[0.102515, 0.007301, 0.005000, 0.000000, 3.141593, -0.000000]),accel_mss,speed_ms,0,0.001)
    |   movel(pose_trans(ref_frame,p[0.103888, 0.005419, 0.005000, -0.000000, 3.141593, -0.000000]),accel_mss,speed_ms,0,0) # end trace
    |   speed_ms    = 0.002
    |   movel(pose_trans(ref_frame,p[0.103888, 0.005419, -0.000125, -0.000000, 3.141593, -0.000000]),accel_mss,speed_ms,0,0) # end trace
    |   speed_ms    = 0.007
    |   movel(pose_trans(ref_frame,p[0.105872, 0.007168, -0.000125, -0.000000, 3.141593, -0.000000]),accel_mss,speed_ms,0,0.001)
    |   movel(pose_trans(ref_frame,p[0.106903, 0.009648, -0.000125, -0.000000, 3.141593, -0.000000]),accel_mss,speed_ms,0,0) # end trace
    |   speed_ms    = 1.000
    |   movel(pose_trans(ref_frame,p[0.106903, 0.009648, 0.005000, -0.000000, 3.141593, 0.000000]),accel_mss,speed_ms,0,0.001)
    |   movel(pose_trans(ref_frame,p[0.060328, 0.029883, 0.005000, -0.000000, 3.141593, -0.000000]),accel_mss,speed_ms,0,0) # end trace
    |   speed_ms    = 0.002
    |   movel(pose_trans(ref_frame,p[0.060328, 0.029883, -0.000125, -0.000000, 3.141593, 0.000000]),accel_mss,speed_ms,0,0) # end trace
    |   speed_ms    = 0.007
    |   movel(pose_trans(ref_frame,p[0.061545, 0.026529, -0.000125, -0.000000, 3.141593, -0.000000]),accel_mss,speed_ms,0,0.001)
    |   movel(pose_trans(ref_frame,p[0.064629, 0.024736, -0.000125, 0.000000, 3.141593, 0.000000]),accel_mss,speed_ms,0,0) # end trace
    |   speed_ms    = 1.000
    |   movel(pose_trans(ref_frame,p[0.064629, 0.024736, 0.005000, 0.000000, 3.141593, -0.000000]),accel_mss,speed_ms,0,0.001)
    |   movel(pose_trans(ref_frame,p[0.057190, 0.026577, 0.005000, 0.000000, 3.141593, 0.000000]),accel_mss,speed_ms,0,0) # end trace
    |   speed_ms    = 0.002
    |   movel(pose_trans(ref_frame,p[0.057190, 0.026577, -0.000125, 0.000000, 3.141593, 0.000000]),accel_mss,speed_ms,0,0) # end trace
    |   speed_ms    = 0.007
    |   movel(pose_trans(ref_frame,p[0.051975, 0.033593, -0.000125, -0.000000, 3.141593, -0.000000]),accel_mss,speed_ms,0,0.001)
    |   movel(pose_trans(ref_frame,p[0.050866, 0.042158, -0.000125, 0.000000, 3.141593, 0.000000]),accel_mss,speed_ms,0,0.001)
    |   movel(pose_trans(ref_frame,p[0.051599, 0.047516, -0.000125, -0.000000, 3.141593, -0.000000]),accel_mss,speed_ms,0,0.001)
    |   movel(pose_trans(ref_frame,p[0.056672, 0.050130, -0.000125, -0.000000, 3.141593, -0.000000]),accel_mss,speed_ms,0,0.001)
    |   movel(pose_trans(ref_frame,p[0.060289, 0.047785, -0.000125, -0.000000, 3.141593, 0.000000]),accel_mss,speed_ms,0,0.001)
    |   movel(pose_trans(ref_frame,p[0.063209, 0.044580, -0.000125, 0.000000, 3.141593, 0.000000]),accel_mss,speed_ms,0,0.001)
    |   movel(pose_trans(ref_frame,p[0.066146, 0.040717, -0.000125, 0.000000, 3.141593, -0.000000]),accel_mss,speed_ms,0,0.001)
    |   movel(pose_trans(ref_frame,p[0.068714, 0.036598, -0.000125, -0.000000, 3.141593, -0.000000]),accel_mss,speed_ms,0,0.001)
    |   movel(pose_trans(ref_frame,p[0.072170, 0.031427, -0.000125, -0.000000, 3.141593, -0.000000]),accel_mss,speed_ms,0,0.001)
    |   movel(pose_trans(ref_frame,p[0.076311, 0.026771, -0.000125, 0.000000, 3.141593, -0.000000]),accel_mss,speed_ms,0,0.001)
    |   movel(pose_trans(ref_frame,p[0.083393, 0.020930, -0.000125, 0.000000, 3.141593, -0.000000]),accel_mss,speed_ms,0,0.001)
    |   movel(pose_trans(ref_frame,p[0.091871, 0.017262, -0.000125, -0.000000, 3.141593, -0.000000]),accel_mss,speed_ms,0,0.001)
    |   movel(pose_trans(ref_frame,p[0.098129, 0.016737, -0.000125, 0.000000, 3.141593, -0.000000]),accel_mss,speed_ms,0,0.001)
    |   movel(pose_trans(ref_frame,p[0.104228, 0.018561, -0.000125, -0.000000, 3.141593, -0.000000]),accel_mss,speed_ms,0,0.001)
    |   movel(pose_trans(ref_frame,p[0.108704, 0.022150, -0.000125, -0.000000, 3.141593, -0.000000]),accel_mss,speed_ms,0,0.001)
    |   movel(pose_trans(ref_frame,p[0.111277, 0.027318, -0.000125, 0.000000, 3.141593, -0.000000]),accel_mss,speed_ms,0,0.001)
    |   movel(pose_trans(ref_frame,p[0.111727, 0.031817, -0.000125, -0.000000, 3.141593, -0.000000]),accel_mss,speed_ms,0,0.001)
    |   movel(pose_trans(ref_frame,p[0.111303, 0.036321, -0.000125, -0.000000, 3.141593, -0.000000]),accel_mss,speed_ms,0,0.001)
    |   movel(pose_trans(ref_frame,p[0.109144, 0.043595, -0.000125, -0.000000, 3.141593, 0.000000]),accel_mss,speed_ms,0,0.001)
    |   movel(pose_trans(ref_frame,p[0.109416, 0.044385, -0.000125, 0.000000, 3.141593, -0.000000]),accel_mss,speed_ms,0,0.001)
    |   movel(pose_trans(ref_frame,p[0.102207, 0.041638, -0.000125, -0.000000, 3.141593, 0.000000]),accel_mss,speed_ms,0,0.001)
    |   movel(pose_trans(ref_frame,p[0.094546, 0.040761, -0.000125, -0.000000, 3.141593, -0.000000]),accel_mss,speed_ms,0,0.001)
    |   movel(pose_trans(ref_frame,p[0.087506, 0.042303, -0.000125, -0.000000, 3.141593, 0.000000]),accel_mss,speed_ms,0,0.001)
    |   movel(pose_trans(ref_frame,p[0.082847, 0.048068, -0.000125, 0.000000, 3.141593, -0.000000]),accel_mss,speed_ms,0,0.001)
    |   movel(pose_trans(ref_frame,p[0.082646, 0.053380, -0.000125, 0.000000, 3.141593, -0.000000]),accel_mss,speed_ms,0,0.001)
    |   movel(pose_trans(ref_frame,p[0.083744, 0.058600, -0.000125, -0.000000, 3.141593, 0.000000]),accel_mss,speed_ms,0,0.001)
    |   movel(pose_trans(ref_frame,p[0.086095, 0.064641, -0.000125, -0.000000, 3.141593, 0.000000]),accel_mss,speed_ms,0,0.001)
    |   movel(pose_trans(ref_frame,p[0.089301, 0.070222, -0.000125, 0.000000, 3.141593, -0.000000]),accel_mss,speed_ms,0,0.001)
    |   movel(pose_trans(ref_frame,p[0.086810, 0.072472, -0.000125, -0.000000, 3.141593, -0.000000]),accel_mss,speed_ms,0,0.001)
    |   movel(pose_trans(ref_frame,p[0.087050, 0.075867, -0.000125, 0.000000, 3.141593, -0.000000]),accel_mss,speed_ms,0,0.001)
    |   movel(pose_trans(ref_frame,p[0.090707, 0.076535, -0.000125, 0.000000, 3.141593, 0.000000]),accel_mss,speed_ms,0,0.001)
    |   movel(pose_trans(ref_frame,p[0.094129, 0.075552, -0.000125, 0.000000, 3.141593, -0.000000]),accel_mss,speed_ms,0,0.001)
    |   movel(pose_trans(ref_frame,p[0.096226, 0.077351, -0.000125, 0.000000, 3.141593, 0.000000]),accel_mss,speed_ms,0,0.001)
    |   movel(pose_trans(ref_frame,p[0.098927, 0.078130, -0.000125, -0.000000, 3.141593, -0.000000]),accel_mss,speed_ms,0,0.001)
    |   movel(pose_trans(ref_frame,p[0.100254, 0.077063, -0.000125, -0.000000, 3.141593, -0.000000]),accel_mss,speed_ms,0,0.001)
    |   movel(pose_trans(ref_frame,p[0.100355, 0.075427, -0.000125, -0.000000, 3.141593, 0.000000]),accel_mss,speed_ms,0,0.001)
    |   movel(pose_trans(ref_frame,p[0.099877, 0.073612, -0.000125, -0.000000, 3.141593, -0.000000]),accel_mss,speed_ms,0,0.001)
    |   movel(pose_trans(ref_frame,p[0.099201, 0.071858, -0.000125, 0.000000, 3.141593, -0.000000]),accel_mss,speed_ms,0,0.001)
    |   movel(pose_trans(ref_frame,p[0.103018, 0.067957, -0.000125, 0.000000, 3.141593, 0.000000]),accel_mss,speed_ms,0,0.001)
    |   movel(pose_trans(ref_frame,p[0.106764, 0.063949, -0.000125, -0.000000, 3.141593, 0.000000]),accel_mss,speed_ms,0,0.001)
    |   movel(pose_trans(ref_frame,p[0.109861, 0.059715, -0.000125, -0.000000, 3.141593, 0.000000]),accel_mss,speed_ms,0,0.001)
    |   movel(pose_trans(ref_frame,p[0.112794, 0.055457, -0.000125, -0.000000, 3.141593, -0.000000]),accel_mss,speed_ms,0,0.001)
    |   movel(pose_trans(ref_frame,p[0.115604, 0.062999, -0.000125, -0.000000, 3.141593, -0.000000]),accel_mss,speed_ms,0,0.001)
    |   movel(pose_trans(ref_frame,p[0.114891, 0.071003, -0.000125, -0.000000, 3.141593, 0.000000]),accel_mss,speed_ms,0,0.001)
    |   movel(pose_trans(ref_frame,p[0.112080, 0.076702, -0.000125, 0.000000, 3.141593, 0.000000]),accel_mss,speed_ms,0,0.001)
    |   movel(pose_trans(ref_frame,p[0.108075, 0.081615, -0.000125, 0.000000, 3.141593, 0.000000]),accel_mss,speed_ms,0,0.001)
    |   movel(pose_trans(ref_frame,p[0.105812, 0.083875, -0.000125, 0.000000, 3.141593, -0.000000]),accel_mss,speed_ms,0,0.001)
    |   movel(pose_trans(ref_frame,p[0.103487, 0.086069, -0.000125, -0.000000, 3.141593, -0.000000]),accel_mss,speed_ms,0,0.001)
    |   movel(pose_trans(ref_frame,p[0.102312, 0.087225, -0.000125, 0.000000, 3.141593, 0.000000]),accel_mss,speed_ms,0,0.001)
    |   movel(pose_trans(ref_frame,p[0.101096, 0.088329, -0.000125, -0.000000, 3.141593, 0.000000]),accel_mss,speed_ms,0,0.001)
    |   movel(pose_trans(ref_frame,p[0.100022, 0.089173, -0.000125, -0.000000, 3.141593, -0.000000]),accel_mss,speed_ms,0,0.001)
    |   movel(pose_trans(ref_frame,p[0.099230, 0.090376, -0.000125, 0.000000, 3.141593, 0.000000]),accel_mss,speed_ms,0,0.001)
    |   movel(pose_trans(ref_frame,p[0.100305, 0.094055, -0.000125, 0.000000, 3.141593, 0.000000]),accel_mss,speed_ms,0,0.001)
    |   movel(pose_trans(ref_frame,p[0.103500, 0.096044, -0.000125, 0.000000, 3.141593, 0.000000]),accel_mss,speed_ms,0,0.001)
    |   movel(pose_trans(ref_frame,p[0.108673, 0.096632, -0.000125, -0.000000, 3.141593, -0.000000]),accel_mss,speed_ms,0,0.001)
    |   movel(pose_trans(ref_frame,p[0.113470, 0.094649, -0.000125, -0.000000, 3.141593, -0.000000]),accel_mss,speed_ms,0,0.001)
    |   movel(pose_trans(ref_frame,p[0.115884, 0.092212, -0.000125, 0.000000, 3.141593, -0.000000]),accel_mss,speed_ms,0,0.001)
    |   movel(pose_trans(ref_frame,p[0.117831, 0.089348, -0.000125, 0.000000, 3.141593, 0.000000]),accel_mss,speed_ms,0,0.001)
    |   movel(pose_trans(ref_frame,p[0.121821, 0.081613, -0.000125, 0.000000, 3.141593, 0.000000]),accel_mss,speed_ms,0,0.001)
    |   movel(pose_trans(ref_frame,p[0.124190, 0.073150, -0.000125, 0.000000, 3.141593, -0.000000]),accel_mss,speed_ms,0,0.001)
    |   movel(pose_trans(ref_frame,p[0.124662, 0.066322, -0.000125, -0.000000, 3.141593, 0.000000]),accel_mss,speed_ms,0,0.001)
    |   movel(pose_trans(ref_frame,p[0.123389, 0.059599, -0.000125, 0.000000, 3.141593, -0.000000]),accel_mss,speed_ms,0,0.001)
    |   movel(pose_trans(ref_frame,p[0.120501, 0.054223, -0.000125, 0.000000, 3.141593, -0.000000]),accel_mss,speed_ms,0,0.001)
    |   movel(pose_trans(ref_frame,p[0.116303, 0.049794, -0.000125, 0.000000, 3.141593, 0.000000]),accel_mss,speed_ms,0,0.001)
    |   movel(pose_trans(ref_frame,p[0.117724, 0.046098, -0.000125, -0.000000, 3.141593, -0.000000]),accel_mss,speed_ms,0,0.001)
    |   movel(pose_trans(ref_frame,p[0.119069, 0.042373, -0.000125, -0.000000, 3.141593, 0.000000]),accel_mss,speed_ms,0,0.001)
    |   movel(pose_trans(ref_frame,p[0.119475, 0.030424, -0.000125, 0.000000, 3.141593, -0.000000]),accel_mss,speed_ms,0,0.001)
    |   movel(pose_trans(ref_frame,p[0.114736, 0.019502, -0.000125, -0.000000, 3.141593, -0.000000]),accel_mss,speed_ms,0,0.001)
    |   movel(pose_trans(ref_frame,p[0.111502, 0.015173, -0.000125, -0.000000, 3.141593, -0.000000]),accel_mss,speed_ms,0,0.001)
    |   movel(pose_trans(ref_frame,p[0.107444, 0.011583, -0.000125, 0.000000, 3.141593, -0.000000]),accel_mss,speed_ms,0,0.001)
    |   movel(pose_trans(ref_frame,p[0.095751, 0.007628, -0.000125, -0.000000, 3.141593, -0.000000]),accel_mss,speed_ms,0,0.001)
    |   movel(pose_trans(ref_frame,p[0.083641, 0.009209, -0.000125, -0.000000, 3.141593, -0.000000]),accel_mss,speed_ms,0,0.001)
    |   movel(pose_trans(ref_frame,p[0.080695, 0.010347, -0.000125, 0.000000, 3.141593, -0.000000]),accel_mss,speed_ms,0,0.001)
    |   movel(pose_trans(ref_frame,p[0.077874, 0.011755, -0.000125, 0.000000, 3.141593, -0.000000]),accel_mss,speed_ms,0,0.001)
    |   movel(pose_trans(ref_frame,p[0.071980, 0.016389, -0.000125, 0.000000, 3.141593, -0.000000]),accel_mss,speed_ms,0,0.001)
    |   movel(pose_trans(ref_frame,p[0.067651, 0.022475, -0.000125, 0.000000, 3.141593, 0.000000]),accel_mss,speed_ms,0,0.001)
    |   movel(pose_trans(ref_frame,p[0.066019, 0.025717, -0.000125, -0.000000, 3.141593, 0.000000]),accel_mss,speed_ms,0,0.001)
    |   movel(pose_trans(ref_frame,p[0.064575, 0.029076, -0.000125, 0.000000, 3.141593, 0.000000]),accel_mss,speed_ms,0,0.001)
    |   movel(pose_trans(ref_frame,p[0.062144, 0.034805, -0.000125, -0.000000, 3.141593, -0.000000]),accel_mss,speed_ms,0,0.001)
    |   movel(pose_trans(ref_frame,p[0.058319, 0.039744, -0.000125, 0.000000, 3.141593, -0.000000]),accel_mss,speed_ms,0,0.001)
    |   movel(pose_trans(ref_frame,p[0.057281, 0.040437, -0.000125, 0.000000, 3.141593, -0.000000]),accel_mss,speed_ms,0,0.001)
    |   movel(pose_trans(ref_frame,p[0.056114, 0.040572, -0.000125, 0.000000, 3.141593, -0.000000]),accel_mss,speed_ms,0,0.001)
    |   movel(pose_trans(ref_frame,p[0.055557, 0.040309, -0.000125, -0.000000, 3.141593, -0.000000]),accel_mss,speed_ms,0,0.001)
    |   movel(pose_trans(ref_frame,p[0.055100, 0.039883, -0.000125, 0.000000, 3.141593, 0.000000]),accel_mss,speed_ms,0,0.001)
    |   movel(pose_trans(ref_frame,p[0.054031, 0.036524, -0.000125, 0.000000, 3.141593, 0.000000]),accel_mss,speed_ms,0,0.001)
    |   movel(pose_trans(ref_frame,p[0.054652, 0.033104, -0.000125, -0.000000, 3.141593, -0.000000]),accel_mss,speed_ms,0,0.001)
    |   movel(pose_trans(ref_frame,p[0.056106, 0.029633, -0.000125, -0.000000, 3.141593, -0.000000]),accel_mss,speed_ms,0,0.001)
    |   movel(pose_trans(ref_frame,p[0.058416, 0.026661, -0.000125, -0.000000, 3.141593, -0.000000]),accel_mss,speed_ms,0,0) # end trace
    |   speed_ms    = 1.000
    |   movel(pose_trans(ref_frame,p[0.058416, 0.026661, 0.005000, -0.000000, 3.141593, -0.000000]),accel_mss,speed_ms,0,0.001)
    |   movel(pose_trans(ref_frame,p[0.058068, 0.033534, 0.005000, -0.000000, 3.141593, 0.000000]),accel_mss,speed_ms,0,0) # end trace
    |   speed_ms    = 0.002
    |   movel(pose_trans(ref_frame,p[0.058068, 0.033534, -0.000125, -0.000000, 3.141593, 0.000000]),accel_mss,speed_ms,0,0) # end trace
    |   speed_ms    = 0.007
    |   movel(pose_trans(ref_frame,p[0.059788, 0.032079, -0.000125, -0.000000, 3.141593, -0.000000]),accel_mss,speed_ms,0,0.001)
    |   movel(pose_trans(ref_frame,p[0.061936, 0.031324, -0.000125, 0.000000, 3.141593, 0.000000]),accel_mss,speed_ms,0,0) # end trace
    |   speed_ms    = 1.000
    |   movel(pose_trans(ref_frame,p[0.061936, 0.031324, 0.005000, 0.000000, 3.141593, -0.000000]),accel_mss,speed_ms,0,0.001)
    |   movel(pose_trans(ref_frame,p[0.055124, 0.036361, 0.005000, 0.000000, 3.141593, -0.000000]),accel_mss,speed_ms,0,0) # end trace
    |   speed_ms    = 0.002
    |   movel(pose_trans(ref_frame,p[0.055124, 0.036361, -0.000125, 0.000000, 3.141593, 0.000000]),accel_mss,speed_ms,0,0) # end trace
    |   speed_ms    = 0.007
    |   movel(pose_trans(ref_frame,p[0.057458, 0.035205, -0.000125, -0.000000, 3.141593, 0.000000]),accel_mss,speed_ms,0,0.001)
    |   movel(pose_trans(ref_frame,p[0.060021, 0.035187, -0.000125, 0.000000, 3.141593, 0.000000]),accel_mss,speed_ms,0,0) # end trace
    |   speed_ms    = 1.000
    |   movel(pose_trans(ref_frame,p[0.060021, 0.035187, 0.005000, 0.000000, 3.141593, -0.000000]),accel_mss,speed_ms,0,0.001)
    |   movel(pose_trans(ref_frame,p[0.037438, 0.051490, 0.005000, -0.000000, 3.141593, -0.000000]),accel_mss,speed_ms,0,0) # end trace
    |   speed_ms    = 0.002
    |   movel(pose_trans(ref_frame,p[0.037438, 0.051490, -0.000125, -0.000000, 3.141593, -0.000000]),accel_mss,speed_ms,0,0) # end trace
    |   speed_ms    = 0.007
    |   movel(pose_trans(ref_frame,p[0.039085, 0.048665, -0.000125, -0.000000, 3.141593, -0.000000]),accel_mss,speed_ms,0,0.001)
    |   movel(pose_trans(ref_frame,p[0.042025, 0.047108, -0.000125, -0.000000, 3.141593, 0.000000]),accel_mss,speed_ms,0,0) # end trace
    |   speed_ms    = 1.000
    |   movel(pose_trans(ref_frame,p[0.042025, 0.047108, 0.005000, -0.000000, 3.141593, -0.000000]),accel_mss,speed_ms,0,0.001)
    |   movel(pose_trans(ref_frame,p[0.037743, 0.054320, 0.005000, -0.000000, 3.141593, 0.000000]),accel_mss,speed_ms,0,0) # end trace
    |   speed_ms    = 0.002
    |   movel(pose_trans(ref_frame,p[0.037743, 0.054320, -0.000125, -0.000000, 3.141593, -0.000000]),accel_mss,speed_ms,0,0) # end trace
    |   speed_ms    = 0.007
    |   movel(pose_trans(ref_frame,p[0.039534, 0.052976, -0.000125, 0.000000, 3.141593, 0.000000]),accel_mss,speed_ms,0,0.001)
    |   movel(pose_trans(ref_frame,p[0.041720, 0.052687, -0.000125, 0.000000, 3.141593, 0.000000]),accel_mss,speed_ms,0,0) # end trace
    |   speed_ms    = 1.000
    |   movel(pose_trans(ref_frame,p[0.041720, 0.052687, 0.005000, 0.000000, 3.141593, -0.000000]),accel_mss,speed_ms,0,0.001)
    |   movel(pose_trans(ref_frame,p[0.034640, 0.054394, 0.005000, -0.000000, 3.141593, 0.000000]),accel_mss,speed_ms,0,0) # end trace
    |   speed_ms    = 0.002
    |   movel(pose_trans(ref_frame,p[0.034640, 0.054394, -0.000125, -0.000000, 3.141593, 0.000000]),accel_mss,speed_ms,0,0) # end trace
    |   speed_ms    = 0.007
    |   movel(pose_trans(ref_frame,p[0.036094, 0.055352, -0.000125, 0.000000, 3.141593, -0.000000]),accel_mss,speed_ms,0,0.001)
    |   movel(pose_trans(ref_frame,p[0.037323, 0.056583, -0.000125, 0.000000, 3.141593, 0.000000]),accel_mss,speed_ms,0,0.001)
    |   movel(pose_trans(ref_frame,p[0.036251, 0.056195, -0.000125, 0.000000, 3.141593, -0.000000]),accel_mss,speed_ms,0,0.001)
    |   movel(pose_trans(ref_frame,p[0.035676, 0.056788, -0.000125, -0.000000, 3.141593, -0.000000]),accel_mss,speed_ms,0,0.001)
    |   movel(pose_trans(ref_frame,p[0.036004, 0.057087, -0.000125, 0.000000, 3.141593, 0.000000]),accel_mss,speed_ms,0,0.001)
    |   movel(pose_trans(ref_frame,p[0.036453, 0.057341, -0.000125, 0.000000, 3.141593, -0.000000]),accel_mss,speed_ms,0,0.001)
    |   movel(pose_trans(ref_frame,p[0.036816, 0.057663, -0.000125, -0.000000, 3.141593, 0.000000]),accel_mss,speed_ms,0,0.001)
    |   movel(pose_trans(ref_frame,p[0.037155, 0.058010, -0.000125, 0.000000, 3.141593, 0.000000]),accel_mss,speed_ms,0,0.001)
    |   movel(pose_trans(ref_frame,p[0.038705, 0.060512, -0.000125, 0.000000, 3.141593, -0.000000]),accel_mss,speed_ms,0,0.001)
    |   movel(pose_trans(ref_frame,p[0.040296, 0.062944, -0.000125, -0.000000, 3.141593, -0.000000]),accel_mss,speed_ms,0,0.001)
    |   movel(pose_trans(ref_frame,p[0.038173, 0.061238, -0.000125, -0.000000, 3.141593, 0.000000]),accel_mss,speed_ms,0,0.001)
    |   movel(pose_trans(ref_frame,p[0.035807, 0.060029, -0.000125, 0.000000, 3.141593, 0.000000]),accel_mss,speed_ms,0,0.001)
    |   movel(pose_trans(ref_frame,p[0.037392, 0.061586, -0.000125, 0.000000, 3.141593, 0.000000]),accel_mss,speed_ms,0,0.001)
    |   movel(pose_trans(ref_frame,p[0.038946, 0.063175, -0.000125, 0.000000, 3.141593, 0.000000]),accel_mss,speed_ms,0,0.001)
    |   movel(pose_trans(ref_frame,p[0.040397, 0.065436, -0.000125, 0.000000, 3.141593, -0.000000]),accel_mss,speed_ms,0,0.001)
    |   movel(pose_trans(ref_frame,p[0.041658, 0.067847, -0.000125, 0.000000, 3.141593, 0.000000]),accel_mss,speed_ms,0,0.001)
    |   movel(pose_trans(ref_frame,p[0.040524, 0.066649, -0.000125, 0.000000, 3.141593, 0.000000]),accel_mss,speed_ms,0,0.001)
    |   movel(pose_trans(ref_frame,p[0.039111, 0.065757, -0.000125, -0.000000, 3.141593, -0.000000]),accel_mss,speed_ms,0,0.001)
    |   movel(pose_trans(ref_frame,p[0.037625, 0.065000, -0.000125, -0.000000, 3.141593, 0.000000]),accel_mss,speed_ms,0,0.001)
    |   movel(pose_trans(ref_frame,p[0.036198, 0.064151, -0.000125, 0.000000, 3.141593, 0.000000]),accel_mss,speed_ms,0,0.001)
    |   movel(pose_trans(ref_frame,p[0.039105, 0.067925, -0.000125, -0.000000, 3.141593, 0.000000]),accel_mss,speed_ms,0,0.001)
    |   movel(pose_trans(ref_frame,p[0.041381, 0.072108, -0.000125, 0.000000, 3.141593, 0.000000]),accel_mss,speed_ms,0,0.001)
    |   movel(pose_trans(ref_frame,p[0.041794, 0.073469, -0.000125, 0.000000, 3.141593, -0.000000]),accel_mss,speed_ms,0,0.001)
    |   movel(pose_trans(ref_frame,p[0.042373, 0.074695, -0.000125, -0.000000, 3.141593, -0.000000]),accel_mss,speed_ms,0,0.001)
    |   movel(pose_trans(ref_frame,p[0.039337, 0.072016, -0.000125, -0.000000, 3.141593, -0.000000]),accel_mss,speed_ms,0,0.001)
    |   movel(pose_trans(ref_frame,p[0.035632, 0.070382, -0.000125, -0.000000, 3.141593, 0.000000]),accel_mss,speed_ms,0,0.001)
    |   movel(pose_trans(ref_frame,p[0.037720, 0.073342, -0.000125, -0.000000, 3.141593, -0.000000]),accel_mss,speed_ms,0,0.001)
    |   movel(pose_trans(ref_frame,p[0.039396, 0.076552, -0.000125, 0.000000, 3.141593, -0.000000]),accel_mss,speed_ms,0,0.001)
    |   movel(pose_trans(ref_frame,p[0.039868, 0.078216, -0.000125, 0.000000, 3.141593, -0.000000]),accel_mss,speed_ms,0,0.001)
    |   movel(pose_trans(ref_frame,p[0.040440, 0.079840, -0.000125, -0.000000, 3.141593, 0.000000]),accel_mss,speed_ms,0,0.001)
    |   movel(pose_trans(ref_frame,p[0.039501, 0.078473, -0.000125, -0.000000, 3.141593, 0.000000]),accel_mss,speed_ms,0,0.001)
    |   movel(pose_trans(ref_frame,p[0.038356, 0.077309, -0.000125, 0.000000, 3.141593, 0.000000]),accel_mss,speed_ms,0,0.001)
    |   movel(pose_trans(ref_frame,p[0.036770, 0.076678, -0.000125, 0.000000, 3.141593, -0.000000]),accel_mss,speed_ms,0,0.001)
    |   movel(pose_trans(ref_frame,p[0.035747, 0.075923, -0.000125, 0.000000, 3.141593, 0.000000]),accel_mss,speed_ms,0,0.001)
    |   movel(pose_trans(ref_frame,p[0.036307, 0.077324, -0.000125, -0.000000, 3.141593, -0.000000]),accel_mss,speed_ms,0,0.001)
    |   movel(pose_trans(ref_frame,p[0.036712, 0.078862, -0.000125, -0.000000, 3.141593, 0.000000]),accel_mss,speed_ms,0,0.001)
    |   movel(pose_trans(ref_frame,p[0.036925, 0.080746, -0.000125, 0.000000, 3.141593, -0.000000]),accel_mss,speed_ms,0,0.001)
    |   movel(pose_trans(ref_frame,p[0.037349, 0.082560, -0.000125, 0.000000, 3.141593, 0.000000]),accel_mss,speed_ms,0,0.001)
    |   movel(pose_trans(ref_frame,p[0.035037, 0.077904, -0.000125, -0.000000, 3.141593, -0.000000]),accel_mss,speed_ms,0,0.001)
    |   movel(pose_trans(ref_frame,p[0.031908, 0.073663, -0.000125, 0.000000, 3.141593, -0.000000]),accel_mss,speed_ms,0,0.001)
    |   movel(pose_trans(ref_frame,p[0.033470, 0.076644, -0.000125, 0.000000, 3.141593, 0.000000]),accel_mss,speed_ms,0,0.001)
    |   movel(pose_trans(ref_frame,p[0.034122, 0.079939, -0.000125, 0.000000, 3.141593, -0.000000]),accel_mss,speed_ms,0,0.001)
    |   movel(pose_trans(ref_frame,p[0.033615, 0.078723, -0.000125, 0.000000, 3.141593, -0.000000]),accel_mss,speed_ms,0,0.001)
    |   movel(pose_trans(ref_frame,p[0.032748, 0.077709, -0.000125, 0.000000, 3.141593, 0.000000]),accel_mss,speed_ms,0,0.001)
    |   movel(pose_trans(ref_frame,p[0.031708, 0.076881, -0.000125, 0.000000, 3.141593, -0.000000]),accel_mss,speed_ms,0,0.001)
    |   movel(pose_trans(ref_frame,p[0.030613, 0.076122, -0.000125, -0.000000, 3.141593, 0.000000]),accel_mss,speed_ms,0,0.001)
    |   movel(pose_trans(ref_frame,p[0.028724, 0.074649, -0.000125, 0.000000, 3.141593, -0.000000]),accel_mss,speed_ms,0,0.001)
    |   movel(pose_trans(ref_frame,p[0.026991, 0.072996, -0.000125, 0.000000, 3.141593, 0.000000]),accel_mss,speed_ms,0,0.001)
    |   movel(pose_trans(ref_frame,p[0.028105, 0.075462, -0.000125, -0.000000, 3.141593, -0.000000]),accel_mss,speed_ms,0,0.001)
    |   movel(pose_trans(ref_frame,p[0.029613, 0.077709, -0.000125, -0.000000, 3.141593, -0.000000]),accel_mss,speed_ms,0,0.001)
    |   movel(pose_trans(ref_frame,p[0.027366, 0.075880, -0.000125, -0.000000, 3.141593, -0.000000]),accel_mss,speed_ms,0,0.001)
    |   movel(pose_trans(ref_frame,p[0.025329, 0.073822, -0.000125, -0.000000, 3.141593, -0.000000]),accel_mss,speed_ms,0,0) # end trace
    |   speed_ms    = 1.000
    |   movel(pose_trans(ref_frame,p[0.025329, 0.073822, 0.005000, -0.000000, 3.141593, 0.000000]),accel_mss,speed_ms,0,0.001)
    |   movel(pose_trans(ref_frame,p[0.022702, 0.069235, 0.005000, -0.000000, 3.141593, -0.000000]),accel_mss,speed_ms,0,0) # end trace
    |   speed_ms    = 0.002
    |   movel(pose_trans(ref_frame,p[0.022702, 0.069235, -0.000125, -0.000000, 3.141593, 0.000000]),accel_mss,speed_ms,0,0) # end trace
    |   speed_ms    = 0.007
    |   movel(pose_trans(ref_frame,p[0.022198, 0.073448, -0.000125, 0.000000, 3.141593, 0.000000]),accel_mss,speed_ms,0,0.001)
    |   movel(pose_trans(ref_frame,p[0.022184, 0.073968, -0.000125, -0.000000, 3.141593, 0.000000]),accel_mss,speed_ms,0,0.001)
    |   movel(pose_trans(ref_frame,p[0.022404, 0.074393, -0.000125, 0.000000, 3.141593, 0.000000]),accel_mss,speed_ms,0,0.001)
    |   movel(pose_trans(ref_frame,p[0.022637, 0.074525, -0.000125, -0.000000, 3.141593, -0.000000]),accel_mss,speed_ms,0,0.001)
